				IF NOT bManualZIsSafe THEN
					TManualCmd.aTAxis[PA_X].Home.Enable := FALSE;
					TManualCmd.aTAxis[PA_Y].Home.Enable := FALSE;
					IF alrJogStep[PA_X] > lrManMaxXYMoveAllowed-0.1 THEN
						TManualCmd.aTAxis[PA_X].MoveBw.Enable := FALSE;
						TManualCmd.aTAxis[PA_X].MoveFw.Enable := FALSE;
					END_IF
					IF alrJogStep[PA_Y] > lrManMaxXYMoveAllowed-0.1 THEN
						TManualCmd.aTAxis[PA_Y].MoveBw.Enable := FALSE;
						TManualCmd.aTAxis[PA_Y].MoveFw.Enable := FALSE;
					END_IF
					IF alrJogStep[PA_Z1] > lrMaxXYMoveAllowed-0.1 THEN
						TManualCmd.aTAxis[PA_Z1].MoveFw.Enable := FALSE;
					END_IF
					IF alrJogStep[PA_Z2] > lrMaxXYMoveAllowed-0.1 THEN
						TManualCmd.aTAxis[PA_Z2].MoveFw.Enable := FALSE;
					END_IF
					TManualCmd.aTAxisPos[PA_X].MoveToTeach.Enable := TManualCmd.aTAxisPos[PA_X].MoveToTeach.Enable AND ABS(TManualCmd.aTAxisPos[PA_X].TeachedPos-aTRobotAxis[PA_X].lrCurrentPos) < lrManMaxXYMoveAllowed-0.1;
					TManualCmd.aTAxisPos[PA_Y].MoveToTeach.Enable := TManualCmd.aTAxisPos[PA_Y].MoveToTeach.Enable AND ABS(TManualCmd.aTAxisPos[PA_Y].TeachedPos-aTRobotAxis[PA_Y].lrCurrentPos) < lrManMaxXYMoveAllowed-0.1;
				END_IF
				bManInterlockOut := NOT bManualZIsSafe;
				TManualCmd.bWeightTableLeftValid := abWeightTableValid[PH_Left];
				TManualCmd.bWeightTableRightValid := abWeightTableValid[PH_Right];
				FOR i :=0 TO C_WEIGHT_TABLE_MAX DO
					TManualCmd.alrWeightTableLeft[i] := alrWeightTable[PH_Left,i];
					TManualCmd.alrWeightTableRight[i] := alrWeightTable[PH_Right,i];
				END_FOR
				FOR iSide:=0 TO 1 DO
					TManualCmd.TResetMotorUseTime[iSide].Enable := TRUE;
					TManualCmd.TResetSpindleUseTime[iSide].Enable := TRUE;
					TManualCmd.alrRatiog2mm[iSide] := alrRatiog2mm[iSide];
					TManualCmd.adwPearlsCounter[iSide] := adwPearlsCounter[iSide];
				END_FOR
				TManualCmd.lrWeightStepOnZ := lrLoadSensorStep;
				TManualCmd.aiDistanceSensor[0] := iContact1Distance;
				TManualCmd.aiDistanceSensor[1] := iContact2Distance;
				TManualCmd.iWeightSensor := iLoadSensorValue;
				CASE sCurrentState.eStep OF
					SP_ManualStp0 :
						FOR iSide:=0 TO 1 DO
							TManualCmd.aTEjectStick[iSide].Enable := TRUE;
							TManualCmd.aTActivateBlowing[iSide ].Enable := TRUE;
							TManualCmd.TActivateAspirationTable[iSide].Activate := abAspirationPearling[iSide];
							TManualCmd.aTStartMotor[iSide].Activate := abStartPearlingMotor[iSide];
							TManualCmd.aTOpenChuck[iSide].Activate := abOpenChuck[iSide];
							TManualCmd.aTEjectStick[iSide].Activate := abActivateEject[iSide];
							TManualCmd.aTActivateBlowing[iSide].Activate := abActivateBlowing[iSide];
							abStartPearlingMotor[iSide] := FALSE;
							TManualCmd.TActivateAspirationTable[iSide].Enable := TRUE;
							TManualCmd.TActivateAspirationTable[iSide].Activate := abAspirationPearling[iSide];
							TManualCmd.aiSpindleSpeedSetpoint[iSide] := aiSpindleManualSpeed[iSide];
							TManualCmd.aTCalibrateWeight[iSide].Activate := FALSE;
							TManualCmd.aiMotorStartedTimeout[iSide] := aiMotorStartedTimeout[iSide];
							TManualCmd.aiMotorStoppedTimeout[iSide] := aiMotorStoppedTimeout[iSide];
							TManualCmd.TResetMotorUseTime[iSide].Activate := FALSE;
							TManualCmd.TResetSpindleUseTime[iSide].Activate := FALSE;
						END_FOR
						FOR iAxis := 0 TO 3 DO
							TManualCmd.aTAxis[iAxis].JogStep := alrJogStep[iAxis];
							TManualCmd.aTAxis[iAxis].Home.Activate := FALSE;
							TManualCmd.aTAxis[iAxis].MoveFw.Activate := FALSE;
							TManualCmd.aTAxis[iAxis].MoveBw.Activate := FALSE;
							TManualCmd.aTAxis[iAxis].Specific.Activate := FALSE;
							TManualCmd.aTAxisPos[iAxis].MoveToTeach.Activate := FALSE;
						END_FOR
						TManualCmd.iCurrentMotorMinTh := iMCRMinThCurrent;
						TManualCmd.iCurrentMotorWarnTh := iMCRWarnThCurrent;
						TManualCmd.iCurrentMotorMaxTh := iMCRMaxThCurrent;
						TManualCmd.TActivateAspirationSharpen.Enable := TRUE;
						TManualCmd.TActivateAspirationSharpen.Activate := bAspirationSharpenOn;
						TManualCmd.TSafe.Activate := FALSE;
						bCalibrationInProgress := FALSE;
						sCurrentState.eStep := SP_ManualStp1;
					SP_ManualStp1:
						IF bStopReq THEN
							sCurrentState.eStatus := MS_Stopped;
						ELSE
							FOR iSide := 0 TO 1 DO
								abStartPearlingMotor[iSide] := TManualCmd.aTStartMotor[iSide].Activate;
								IF TManualCmd.TResetMotorUseTime[iSide].Activate THEN
									aTMotorCounter[iSide](bReset := TRUE);
									TManualCmd.TResetMotorUseTime[iSide].Activate := FALSE;
								END_IF
								IF TManualCmd.TResetSpindleUseTime[iSide].Activate THEN
									aTSpindleCounter[iSide](bReset := TRUE);
									TManualCmd.TResetSpindleUseTime[iSide].Activate := FALSE;
								END_IF
								IF TManualCmd.aiSpindleSpeedSetpoint[iSide] <> aiSpindleManualSpeed[iSide] THEN
									aiSpindleManualSpeed[iSide] := TManualCmd.aiSpindleSpeedSetpoint[iSide];
								END_IF
								IF TManualCmd.aiMotorStartedTimeout[iSide] <> aiMotorStartedTimeout[iSide] THEN
									aiMotorStartedTimeout[iSide] := TManualCmd.aiMotorStartedTimeout[iSide];
								END_IF
								IF TManualCmd.aiMotorStoppedTimeout[iSide] <> aiMotorStoppedTimeout[iSide] THEN
									aiMotorStoppedTimeout[iSide] := TManualCmd.aiMotorStoppedTimeout[iSide];
								END_IF
								// Calibration
								IF TManualCmd.aTCalibrateWeight[iSide].Activate THEN
									TManualCmd.aTCalibrateWeight[iSide].Activate := FALSE;
									bCalibrationInProgress := TRUE;
									iCurrentManAxis := iSide;
									sCurrentState.eStep := SP_ManualStp20;
								END_IF
							END_FOR
							IF TManualCmd.iCurrentMotorMinTh <> iMCRMinThCurrent THEN
								iMCRMinThCurrent := TManualCmd.iCurrentMotorMinTh;
							END_IF
							IF TManualCmd.iCurrentMotorMaxTh <> iMCRMaxThCurrent THEN
								iMCRMaxThCurrent := TManualCmd.iCurrentMotorMaxTh;
							END_IF
							IF TManualCmd.iCurrentMotorWarnTh <> iMCRWarnThCurrent THEN
								iMCRWarnThCurrent := TManualCmd.iCurrentMotorWarnTh;
							END_IF
							FOR iAxis := 0 TO 3 DO
								TManualCmd.aTAxisPos[iAxis].TeachedPos := alrRobotPos[iAxis,TManualCmd.e_TeachPos];
								IF TManualCmd.aTAxisPos[iAxis].Teach THEN
									alrRobotPos[iAxis,TManualCmd.e_TeachPos] := aTRobotAxis[iAxis].lrCurrentPos;
								END_IF
								TManualCmd.aTAxisPos[iAxis].Teach := FALSE;
							END_FOR
							FOR iAxis := 0 TO 3 DO
								IF (alrJogStep[iAxis] <> TManualCmd.aTAxis[iAxis].JogStep) THEN
									alrJogStep[iAxis] := TManualCmd.aTAxis[iAxis].JogStep;
								END_IF
								IF TManualCmd.aTAxisPos[iAxis].MoveToTeach.Activate THEN
									alrTargetPos[iAxis] := TManualCmd.aTAxisPos[iAxis].TeachedPos;
									iCurrentManAxis := iAxis;
									sCurrentState.eStep := SP_ManualStp2;
									EXIT;
								END_IF
								IF TManualCmd.aTAxis[iAxis].MoveFw.Activate THEN
									alrTargetPos[iAxis] := aTRobotAxis[iAxis].lrCurrentPos + alrJogStep[iAxis];
									iCurrentManAxis := iAxis;
									sCurrentState.eStep := SP_ManualStp2;
									EXIT;
								END_IF
								IF TManualCmd.aTAxis[iAxis].MoveBw.Activate THEN
									alrTargetPos[iAxis] := aTRobotAxis[iAxis].lrCurrentPos - alrJogStep[iAxis];
									iCurrentManAxis := iAxis;
									sCurrentState.eStep := SP_ManualStp2;
									EXIT;
								END_IF
								IF TManualCmd.aTAxis[iAxis].Home.Activate THEN
									iCurrentManAxis := iAxis;
									sCurrentState.eStep := SP_ManualStp40;
									EXIT;
								END_IF
							END_FOR
							IF TManualCmd.aTAxis[2].Specific.Activate THEN
								alrTargetPos[PA_Z1] := alrSafePos[PA_Z1];
								iCurrentManAxis := 2;
								sCurrentState.eStep := SP_ManualStp2;
							END_IF
							IF TManualCmd.aTAxis[3].Specific.Activate THEN
								alrTargetPos[PA_Z2] := alrSafePos[PA_Z2];
								iCurrentManAxis := 3;
								sCurrentState.eStep := SP_ManualStp2;
							END_IF
							IF TManualCmd.TSafe.Activate AND  (sCurrentState.eStep = SP_ManualStp1) THEN
								TManualCmd.TSafe.Activate := FALSE;
								sCurrentState.eStep := SP_ManualStp10;
							END_IF
							IF (sCurrentState.eStep = SP_ManualStp1) AND NOT bBypassMCR THEN
								sCurrentState.eStep := SP_ManualStp45;
							END_IF
						END_IF
					SP_ManualStp2:
						aeMoveRobotCommand[iCurrentManAxis] := AC_MoveAtAbsPos;
						sCurrentState.eStep := SP_ManualStp3;
					SP_ManualStp3:
						(* Wait until position is reached *)
						IF (aTRobotAxis[iCurrentManAxis].eCurrentState = AS_InPosition) THEN
							TManualCmd.aTAxisPos[iCurrentManAxis].MoveToTeach.Activate := FALSE;
							TManualCmd.aTAxis[iCurrentManAxis].Home.Activate := FALSE;
							TManualCmd.aTAxis[iCurrentManAxis].MoveFw.Activate := FALSE;
							TManualCmd.aTAxis[iCurrentManAxis].MoveBw.Activate := FALSE;
							TManualCmd.aTAxis[iCurrentManAxis].Specific.Activate := FALSE;
							sCurrentState.eStep := SP_ManualStp1;
						END_IF
					SP_ManualStp10: (*Move  Z1 and Z2 to Limit*)
						aeMoveRobotCommand[PA_Z1] := AC_MoveLimitNeg;
						aeMoveRobotCommand[PA_Z2] := AC_MoveLimitNeg;
						sCurrentState.eStep := SP_ManualStp11;
					SP_ManualStp11:
						IF aTRobotAxis[PA_Z1].eCurrentState= AS_OnLimitNeg AND aTRobotAxis[PA_Z2].eCurrentState= AS_OnLimitNeg THEN
							sCurrentState.eStep := SP_ManualStp12;
						ELSIF (aTRobotAxis[PA_Z1].eCurrentState= AS_OnLimitNeg AND aTRobotAxis[PA_Z2].eCurrentState = AS_InError) OR
							    (aTRobotAxis[PA_Z1].eCurrentState= AS_InError AND aTRobotAxis[PA_Z2].eCurrentState = AS_OnLimitNeg) OR
							    (aTRobotAxis[PA_Z1].eCurrentState= AS_InError AND aTRobotAxis[PA_Z2].eCurrentState = AS_InError) THEN
							sCurrentState.eStep := SP_ManualStp1;
						END_IF
					SP_ManualStp12: (* Init X/Y  *)
						aeMoveRobotCommand[PA_X] := AC_Init;
						aeMoveRobotCommand[PA_Y] := AC_Init;
						sCurrentState.eStep := SP_ManualStp13;
					SP_ManualStp13:
						IF aTRobotAxis[PA_X].eCurrentState= AS_InPosition AND aTRobotAxis[PA_Y].eCurrentState = AS_InPosition THEN
							sCurrentState.eStep := SP_ManualStp14;
						ELSIF (aTRobotAxis[PA_X].eCurrentState= AS_InPosition AND aTRobotAxis[PA_Y].eCurrentState = AS_InError) OR
								(aTRobotAxis[PA_X].eCurrentState= AS_InError AND aTRobotAxis[PA_Y].eCurrentState = AS_InPosition) OR
								(aTRobotAxis[PA_X].eCurrentState= AS_InError AND aTRobotAxis[PA_Y].eCurrentState = AS_InError) THEN
							sCurrentState.eStep := SP_ManualStp1;
						END_IF
					SP_ManualStp14: (* Move X/Y *)
						aeMoveRobotCommand[PA_X] := AC_MoveAtAbsPos;
						aeMoveRobotCommand[PA_Y] := AC_MoveAtAbsPos;
						alrTargetPos[PA_X] := alrSafePos[PA_X];
						alrTargetPos[PA_Y] := alrSafePos[PA_Y];
						sCurrentState.eStep := SP_ManualStp15;
					SP_ManualStp15:
						IF aTRobotAxis[PA_X].eCurrentState= AS_InPosition AND aTRobotAxis[PA_Y].eCurrentState = AS_InPosition THEN
							sCurrentState.eStep := SP_ManualStp16;
						ELSIF (aTRobotAxis[PA_X].eCurrentState= AS_InPosition AND aTRobotAxis[PA_Y].eCurrentState = AS_InError) OR
								(aTRobotAxis[PA_X].eCurrentState= AS_InError AND aTRobotAxis[PA_Y].eCurrentState = AS_InPosition) OR
								(aTRobotAxis[PA_X].eCurrentState= AS_InError AND aTRobotAxis[PA_Y].eCurrentState = AS_InError) THEN
							sCurrentState.eStep := SP_ManualStp1;
						END_IF
					SP_ManualStp16: (* Init Z1 and Z2*)
						aeMoveRobotCommand[PA_Z1] := AC_Init;
						aeMoveRobotCommand[PA_Z2] := AC_Init;
						sCurrentState.eStep := SP_ManualStp17;
					SP_ManualStp17:
						IF aTRobotAxis[PA_Z1].eCurrentState= AS_InPosition AND aTRobotAxis[PA_Z2].eCurrentState = AS_InPosition THEN
							sCurrentState.eStep := SP_ManualStp18;
						ELSIF (aTRobotAxis[PA_Z1].eCurrentState= AS_InPosition AND aTRobotAxis[PA_Z2].eCurrentState = AS_InError) OR
								(aTRobotAxis[PA_Z1].eCurrentState= AS_InError AND aTRobotAxis[PA_Z2].eCurrentState = AS_InPosition) OR
								(aTRobotAxis[PA_Z1].eCurrentState= AS_InError AND aTRobotAxis[PA_Z2].eCurrentState = AS_InError) THEN
							sCurrentState.eStep := SP_ManualStp1;
						END_IF
					SP_ManualStp18: (* Move up Z1 and Z2 *)
						aeMoveRobotCommand[PA_Z1] := AC_MoveAtAbsPos;
						aeMoveRobotCommand[PA_Z2] := AC_MoveAtAbsPos;
						alrTargetPos[PA_Z1] := alrSafePos[PA_Z1];
						alrTargetPos[PA_Z2] := alrSafePos[PA_Z2];
						sCurrentState.eStep := SP_ManualStp19;
					SP_ManualStp19:
						IF (aTRobotAxis[PA_Z1].eCurrentState= AS_InPosition OR aTRobotAxis[PA_Z1].eCurrentState = AS_InError) AND
								(aTRobotAxis[PA_Z2].eCurrentState= AS_InPosition OR aTRobotAxis[PA_Z2].eCurrentState = AS_InError) THEN
							sCurrentState.eStep := SP_ManualStp1;
						END_IF
					SP_ManualStp20:	 (* Do calibration *)
						abStartPearlingMotor[iCurrentManAxis] := FALSE;
						TManualCmd.aTStartMotor[iSide].Activate := FALSE;
						abWeightTableValid[iCurrentManAxis] := FALSE;
						FOR iSide := 0 TO 1 DO		// put the 2 brushes at Z safe position
							alrTargetPos[PA_Z1+iSide] := alrSafePos[PA_Z1+iSide];
							aeMoveRobotCommand[PA_Z1+iSide] := AC_MoveAtAbsPos;
						END_FOR
						sCurrentState.eStep := SP_ManualStp21;
					SP_ManualStp21:
						(* Wait until position is reached *)
						//IF (aTRobotAxis[PA_Z1+iCurrentManAxis].eCurrentState = AS_InPosition) AND aTWaitMotorStopped[iCurrentManAxis].Q THEN
						IF (aTRobotAxis[PA_Z1].eCurrentState = AS_InPosition) AND (aTRobotAxis[PA_Z2].eCurrentState = AS_InPosition) AND aTWaitMotorStopped[iCurrentManAxis].Q THEN
							aTStickContactValidated[iCurrentManAxis](IN := FALSE);
							alrLoadSensorOffset[iCurrentManAxis] := iLoadSensorValue;
							aeProbingArea[iCurrentManAxis] := PA_WeightCalibration;
							(* Move to load sensor position *)
							alrTargetPos[PA_X] := alrRobotPos[PA_X, PTP_WeightCalibrationPosZ1+iCurrentManAxis];
							alrTargetPos[PA_Y] := alrRobotPos[PA_Y, PTP_WeightCalibrationPosZ1+iCurrentManAxis];
							aeMoveRobotCommand[PA_X] := AC_MoveAtAbsPos;
							aeMoveRobotCommand[PA_Y] := AC_MoveAtAbsPos;
							sCurrentState.eStep := SP_ManualStp22;
						END_IF
					SP_ManualStp22:
						IF (eRobotXYStatus = AS_InPosition) THEN
							aTStickContactValidated[iCurrentManAxis](IN := TRUE,PT := TStickContactValidTime);
							IF aTStickContactValidated[iCurrentManAxis].Q THEN
								(* Get sensor threshold before getting down, so we can detetced if there is a stick *)
								aiContactThresholdArea[iCurrentManAxis , aeProbingArea[iCurrentManAxis]] := aiContactDistance[iCurrentManAxis];
								alrProbingLimit[iCurrentManAxis] :=  alrRobotPos[PA_Z1+iCurrentManAxis, PTP_WeightCalibrationPosZ1+iCurrentManAxis] + 0.5;
								alrTargetPos[PA_Z1+iCurrentManAxis] := alrRobotPos[PA_Z1+iCurrentManAxis, PTP_WeightCalibrationPosZ1+iCurrentManAxis];
								aeMoveRobotCommand[PA_Z1+iCurrentManAxis] := AC_MoveAtAbsPos;
								sCurrentState.eStep := SP_ManualStp23;
							END_IF
						END_IF
					SP_ManualStp23:
						(* Continuous move probing with analog sensor *)
						IF (aTRobotAxis[PA_Z1+ iCurrentManAxis].eCurrentState = AS_InPosition) THEN
							(* Move 0.5 mm above probing pos to check default sensor value *)
							alrTargetPos[PA_Z1 + iCurrentManAxis] := alrTargetPos[PA_Z1 + iCurrentManAxis] - 0.5;
							alrCurrentSpeed[PA_Z1 + iCurrentManAxis] := alrMaxRobotSpeed[PA_Z1 + iCurrentManAxis];
							aeMoveRobotCommand[PA_Z1 + iCurrentManAxis] := AC_MoveAtAbsPos;
							aTStickContactValidated[iCurrentManAxis](IN := FALSE);
							sCurrentState.eStep := SP_ManualStp24;
						ELSIF (aiContactDistance[iCurrentManAxis] > aiContactThresholdArea[iCurrentManAxis , aeProbingArea[iCurrentManAxis]] + alrSensorRate[iCurrentManAxis] * 0.5) THEN
							(* Stick is present, abort the process *)
							aeMoveRobotCommand[PA_Z1+iCurrentManAxis] := AC_Stop;
							bSecurityError := TRUE;
							iDebugPos := 6;
							iDebugSide := iCurrentManAxis;
							bCalibrationInProgress := FALSE;
							sCurrentState.eStep := SP_ManualStp1;
						END_IF
					SP_ManualStp24:
						IF (aTRobotAxis[PA_Z1 + iCurrentManAxis].eCurrentState = AS_InPosition) THEN
							aTStickContactValidated[iCurrentManAxis](IN := TRUE,PT := TStickContactValidTime);
							IF aTStickContactValidated[iCurrentManAxis].Q THEN
								aiContactThresholdArea[iCurrentManAxis , aeProbingArea[iCurrentManAxis]] := aiContactDistance[iCurrentManAxis];
								(* Move down slowly until we get contact *)
								alrTargetPos[PA_Z1 + iCurrentManAxis] := alrProbingLimit[iCurrentManAxis];
								alrCurrentSpeed[PA_Z1 + iCurrentManAxis] := lrSensorZSpeed;
								aeMoveRobotCommand[PA_Z1 + iCurrentManAxis] := AC_MoveAtAbsPos;
								sCurrentState.eStep := SP_ManualStp25;
							END_IF
						END_IF
					SP_ManualStp25:
						IF (aiContactDistance[iCurrentManAxis] >aiContactThresholdArea[iCurrentManAxis , aeProbingArea[iCurrentManAxis]] + alrSensorRate[iCurrentManAxis] * lrProbingThreshold) THEN
							aTStickContactValidated[iCurrentManAxis](IN := FALSE);
							aeMoveRobotCommand[PA_Z1 + iCurrentManAxis] := AC_Stop;
							sCurrentState.eStep := SP_ManualStp26;
						ELSIF (aTRobotAxis[PA_Z1 + iCurrentManAxis].eCurrentState = AS_InPosition) THEN
							aeMoveRobotCommand[PA_Z1+iCurrentManAxis] := AC_Stop;
							bSecurityError := TRUE;
							iDebugPos := 7;
							iDebugSide := iCurrentManAxis;
							bCalibrationInProgress := FALSE;
							sCurrentState.eStep := SP_ManualStp1;
						END_IF
					SP_ManualStp26:
						IF (aTRobotAxis[PA_Z1 + iCurrentManAxis].eCurrentState = AS_InPosition) THEN
							aTStickContactValidated[iCurrentManAxis](IN := TRUE,PT := TStickContactValidTime);
							IF aTStickContactValidated[iCurrentManAxis].Q THEN
								alrProbingPos[iCurrentManAxis] := aTRobotAxis[PA_Z1 + iCurrentManAxis].lrCurrentPos - (aiContactDistance[iCurrentManAxis] - aiContactThresholdArea[iCurrentManAxis , aeProbingArea[iCurrentManAxis]])/alrSensorRate[iCurrentManAxis];
								(* Move 2 mm above probing pos to check 1st measure *)
								alrTargetPos[PA_Z1 + iCurrentManAxis] := aTRobotAxis[PA_Z1 + iCurrentManAxis].lrCurrentPos - 2;
								alrCurrentSpeed[PA_Z1 + iCurrentManAxis] := alrMaxRobotSpeed[PA_Z1 + iCurrentManAxis];
								aeMoveRobotCommand[PA_Z1 + iCurrentManAxis] := AC_MoveAtAbsPos;
								sCurrentState.eStep := SP_ManualStp27;
							END_IF
						END_IF
					SP_ManualStp27:
						IF (aTRobotAxis[PA_Z1 + iCurrentManAxis].eCurrentState = AS_InPosition) THEN
							(* Move to contact position *)
							alrTargetPos[PA_Z1 + iCurrentManAxis] := alrTargetPos[PA_Z1 + iCurrentManAxis]+2;
							aeMoveRobotCommand[PA_Z1 + iCurrentManAxis] := AC_MoveAtAbsPos;
							aTStickContactValidated[iCurrentManAxis](IN := FALSE);
							sCurrentState.eStep := SP_ManualStp28;
						END_IF
					SP_ManualStp28:
						IF (aTRobotAxis[PA_Z1 + iCurrentManAxis].eCurrentState = AS_InPosition) THEN
							aTStickContactValidated[iCurrentManAxis](IN := TRUE,PT := TStickContactValidTime);
							IF aTStickContactValidated[iCurrentManAxis].Q THEN
								alrCheckProbingPos[iCurrentManAxis] := aTRobotAxis[PA_Z1 + iCurrentManAxis].lrCurrentPos - (aiContactDistance[iCurrentManAxis] - aiContactThresholdArea[iCurrentManAxis , aeProbingArea[iCurrentManAxis]])/alrSensorRate[iCurrentManAxis];
								IF (ABS(alrProbingPos[iCurrentManAxis] - alrCheckProbingPos[iCurrentManAxis]) < 0.05) AND (ABS(alrProbingPos[iCurrentManAxis] -  alrRobotPos[PA_Z1+iCurrentManAxis, PTP_WeightCalibrationPosZ1+iCurrentManAxis]) < 0.5) THEN
									sCurrentState.eStep := SP_ManualStp29;
								ELSE
									bSecurityError := TRUE;
									iDebugPos := 8;
									iDebugSide := iCurrentManAxis;
									bCalibrationInProgress := FALSE;
									sCurrentState.eStep := SP_ManualStp1;
								END_IF
							END_IF
						END_IF
					SP_ManualStp29:
						aTStickContactValidated[iCurrentManAxis](IN := FALSE);
						iTableIndex := 0;
						lrBasePos := alrProbingPos[iCurrentManAxis] - lrWeightCalibrationStartOffsetZ;
						alrTargetPos[PA_Z1+iCurrentManAxis] := lrBasePos;
						alrCurrentSpeed[PA_Z1+iCurrentManAxis] := lrSensorZSpeed;
						aeMoveRobotCommand[PA_Z1+iCurrentManAxis] := AC_MoveAtAbsPos;
						sCurrentState.eStep := SP_ManualStp30;
					SP_ManualStp30:
						IF (aTRobotAxis[PA_Z1+iCurrentManAxis].eCurrentState = AS_InPosition) THEN
							(* Measure delta contact position*)
							aTStickContactValidated[iCurrentManAxis](IN := TRUE,PT := TStickContactValidTime);
							IF aTStickContactValidated[iCurrentManAxis].Q THEN
								alrWeightTable[iCurrentManAxis,iTableIndex] := (INT_TO_LREAL(iLoadSensorValue) - alrLoadSensorOffset[iCurrentManAxis]) / lrLoadSensorRate;
								IF (iTableIndex < C_WEIGHT_TABLE_MAX) THEN
									iTableIndex := iTableIndex+1;
									alrTargetPos[PA_Z1+iCurrentManAxis] := lrBasePos + INT_TO_LREAL(iTableIndex)*lrLoadSensorStep;
									aeMoveRobotCommand[PA_Z1+iCurrentManAxis] := AC_MoveAtAbsPos;
									aTStickContactValidated[iCurrentManAxis](IN := FALSE);
								ELSE
									(* Calculate g to mm ratio *)
									alrRatiog2mm[iCurrentManAxis] := 1/((alrWeightTable[iCurrentManAxis,C_WEIGHT_TABLE_MAX] - alrWeightTable[iCurrentManAxis,10])/((C_WEIGHT_TABLE_MAX - 10)*lrLoadSensorStep));
									(* Move up to safe *)
									alrTargetPos[PA_Z1+iCurrentManAxis] := alrSafePos[PA_Z1+iCurrentManAxis];
									alrCurrentSpeed[PA_Z1+iCurrentManAxis] := alrMaxRobotSpeed[PA_Z1+iCurrentManAxis];
									aeMoveRobotCommand[PA_Z1+iCurrentManAxis] := AC_MoveAtAbsPos;
									sCurrentState.eStep := SP_ManualStp31;
								END_IF
							END_IF
						END_IF
					SP_ManualStp31:
						IF (aTRobotAxis[PA_Z1+iCurrentManAxis].eCurrentState = AS_InPosition) THEN
							abWeightTableValid[iCurrentManAxis] := TRUE;
							bCalibrationInProgress := FALSE;
							sCurrentState.eStep := SP_ManualStp1;
						END_IF
					SP_ManualStp40 : (* Init axis *)
						aeMoveRobotCommand[iCurrentManAxis] := AC_Home;
						sCurrentState.eStep := SP_ManualStp41;
					SP_ManualStp41 : (* Rotate the turn over to go to index position *)
						CASE aTRobotAxis[iCurrentManAxis].eCurrentState OF
							AS_InPosition, AS_InError:
								FOR iAxis := 0 TO 4 DO
									TManualCmd.aTAxis[iCurrentManAxis].Home.Activate := FALSE;
									TManualCmd.aTAxis[iCurrentManAxis].MoveFw.Activate := FALSE;
									TManualCmd.aTAxis[iCurrentManAxis].MoveBw.Activate := FALSE;
								END_FOR
								sCurrentState.eStep := SP_ManualStp1;
						END_CASE
					SP_ManualStp45:
						IF bMCRReady THEN
							yMCRChannel := 1;
							sCurrentState.eStep := SP_ManualStp46;
						END_IF
					SP_ManualStp46:
						(* Read speed *)
						eMCRCommand := MCRC_ReadSpeed;
						sCurrentState.eStep := SP_ManualStp47;
					SP_ManualStp47:
						IF bMCRReady THEN
							TManualCmd.aiMotorSpeed[yMCRChannel-1] := TMCRDrv.iSpeed;
							IF yMCRChannel = 1 THEN
								yMCRChannel := 2;
								sCurrentState.eStep := SP_ManualStp46;
							ELSE
								yMCRChannel := 1;
								sCurrentState.eStep := SP_ManualStp48;
							END_IF
						END_IF
					SP_ManualStp48:
						(* Read current *)
						eMCRCommand := MCRC_ReadCurrent;
						sCurrentState.eStep := SP_ManualStp49;
					SP_ManualStp49:
						IF bMCRReady THEN
							TManualCmd.arMotorCurrent[yMCRChannel-1] := LREAL_TO_REAL(TMCRDrv.lrCurrent);
							IF yMCRChannel = 1 THEN
								yMCRChannel := 2;
								sCurrentState.eStep := SP_ManualStp48;
							ELSE
								yMCRChannel := 1;
								sCurrentState.eStep := SP_ManualStp50;
							END_IF
						END_IF
					SP_ManualStp50:
						(* Set Ratio*)
						eMCRCommand := MCRC_SetRatio;
						TMCRDrv.lrRatio := asStickDataMMI[yMCRChannel - 1].lrMCRRatio;
						sCurrentState.eStep := SP_ManualStp51;
					SP_ManualStp51:
						IF bMCRReady THEN
							IF yMCRChannel = 1 THEN
								yMCRChannel := 2;
								sCurrentState.eStep := SP_ManualStp50;
							ELSE
								yMCRChannel := 1;
								sCurrentState.eStep := SP_ManualStp52;
							END_IF
						END_IF
					SP_ManualStp52:
						(* Set Speed*)
						eMCRCommand := MCRC_SetSpeed;
						TMCRDrv.iSpeedSetpoint := TManualCmd.aiSpindleSpeedSetpoint[yMCRChannel - 1];
						sCurrentState.eStep := SP_ManualStp53;
					SP_ManualStp53:
						IF bMCRReady THEN
							IF yMCRChannel = 1 THEN
								yMCRChannel := 2;
								sCurrentState.eStep := SP_ManualStp52;
							ELSE
								yMCRChannel := 1;
								sCurrentState.eStep := SP_ManualStp54;
							END_IF
						END_IF
					SP_ManualStp54:
						(* Set Parameter*)
						eMCRCommand := MCRC_SetParam;
						TMCRDrv.iOffsetCurrent := iMCROffsetCurrent[yMCRChannel - 1];
						TMCRDrv.iCurrentRatio := iMCRCurrentRatio[yMCRChannel - 1];
						sCurrentState.eStep := SP_ManualStp55;
					SP_ManualStp55:
						IF bMCRReady THEN
							IF yMCRChannel = 1 THEN
								yMCRChannel := 2;
								sCurrentState.eStep := SP_ManualStp54;
							ELSE
								yMCRChannel := 1;
								sCurrentState.eStep := SP_ManualStp1;
							END_IF
						END_IF
				END_CASE
				FOR iSide := 0 TO 1 DO
					abOpenChuck[iSide] := TManualCmd.aTOpenChuck[iSide].Activate;
					abActivateEject[iSide] := TManualCmd.aTEjectStick[iSide].Activate;
					abActivateBlowing[iSide] := TManualCmd.aTActivateBlowing[iSide].Activate;
					abAspirationPearling[iSide] := TManualCmd.TActivateAspirationTable[iSide].Activate;
				END_FOR
				bAspirationSharpenOn := TManualCmd.TActivateAspirationSharpen.Activate;
			MS_Paused:
				IF bStopReq THEN
					sCurrentState.eStatus := MS_Ready;
					sCurrentState.eStep := SP_RunStp1;
				END_IF
		END_CASE
	MC_Init :
		IF sCurrentState.bInitDone THEN
			sCurrentState.eStep := SP_InitStp50;
		ELSE
			sCurrentState.eStep := SP_InitStp1;
		END_IF
		sCurrentState.eStatus := MS_Init;
	MC_Run :
		IF (sCurrentState.eStep = SP_RunStp91) THEN
			sCurrentState.eStep := SP_RunStp92;
		END_IF
		sCurrentState.eStatus := MS_Running;
	MC_Manual :
		sCurrentState.bInitDone := FALSE;
		sCurrentState.eStatus := MS_Manual;
		sCurrentState.eStep := SP_ManualStp0;
	MC_Stop :
		//eMCRCommand := MCRC_UpdateMemory;				// TODO : HFO, Problème de comunication, impossible de mettre à jour les chips, controle si ok?
		sCurrentState.eStatus := MS_Stopped;
END_CASE;

(* The pearling motor doesn't run if not in production *)
IF (sCurrentState.eStatus <> MS_Running) AND (sCurrentState.eStatus <> MS_Manual) THEN
	FOR iSide := 0 TO 1 DO
		abStartPearlingMotor[iSide] := FALSE;
		abActivateBlowing[iSide] := FALSE;
	END_FOR
END_IF
IF (sCurrentState.eStatus = MS_Running) THEN
	FOR iSide:=0 TO 1 DO
		(* Force motor running if possible *)
		IF NOT abDoProbing[iSide] AND NOT abChangeStick[iSide]  AND NOT  abSharpenStick[iSide] AND abChuckClosed[iSide] AND
				((sCurrentState.eStep < SP_RunStp30) OR
				(sCurrentState.eStep > SP_RunStp33)) THEN
			IF bKeepBothHeadWarm THEN
				abStartPearlingMotor[iSide] := TRUE;
			ELSE
				abStartPearlingMotor[iSide] := abUseSpindle[iSide];
			END_IF
		END_IF
	END_FOR
	FOR iSide:=0 TO 1 DO
		abActivateBlowing[iSide] := abStartPearlingMotor[PH_Left] OR abStartPearlingMotor[PH_Right]; (* Activate blowing if at least one head is pearling *)
	END_FOR
END_IF

IF bResetErrors THEN
	sCurrentState.bInError := FALSE;
END_IF

(* Define dynamics *)

FOR iAxis:=0 TO 3 DO
	IF (aeMoveRobotCommand[iAxis] = AC_MoveAtAbsPos) THEN
		IF (ABS(aTRobotAxis[iAxis].lrCurrentPos - alrTargetPos[iAxis]) > 10) THEN
			alrDynParams[iAxis] := alrLowDynParams[iAxis];
		ELSE
			alrDynParams[iAxis] := alrHighDynParams[iAxis];
		END_IF
	END_IF
END_FOR


IF ((ABS(aTRobotAxis[PA_X].lrCurrentPos - alrTargetPos[PA_X]) > lrMaxXYMoveAllowed) AND (aeMoveRobotCommand[PA_X] <> AC_None)) OR
		((ABS(aTRobotAxis[PA_Y].lrCurrentPos - alrTargetPos[PA_Y]) > lrMaxXYMoveAllowed) AND (aeMoveRobotCommand[PA_Y] <> AC_None)) THEN
	IF (aTRobotAxis[PA_Z1].lrCurrentPos > (alrSafePos[PA_Z1] + lrSafeTolerance)) OR
			(aTRobotAxis[PA_Z2].lrCurrentPos > (alrSafePos[PA_Z2] + lrSafeTolerance)) THEN
		IF eStickStep<> SP_RunStp61 AND eStickStep<> SP_RunStp62 THEN
			aeMoveRobotCommand[PA_X] := AC_ForceStop;
			aeMoveRobotCommand[PA_Y] := AC_ForceStop;
			sCurrentState.bInitDone := FALSE;
			bSecurityError := TRUE;
			iDebugPos := 9;
			iDebugSide := -1;
		END_IF
	END_IF
END_IF

IF (sCurrentState.eStatus = MS_Manual) THEN
	FOR iAxis:=0 TO 3 DO
		IF bManualZIsSafe THEN
			alrCurrentSpeed[iAxis] := aTRobotAxis[iAxis].lrFastManualSpeed;
		ELSE
			alrCurrentSpeed[iAxis] :=  aTRobotAxis[iAxis].lrManualSpeed;
		END_IF
	END_FOR
END_IF

(* Robot command *)
aTRobotAxis[PA_X](
	eCommand 		:= aeMoveRobotCommand[PA_X],
	lrTargetPos 		:= alrTargetPos[PA_X],
	lrTargetSpeed 	:= alrCurrentSpeed[PA_X],
	lrAcceleration 	:= alrDynParams[PA_X].Acc,
	lrDeceleration 	:= alrDynParams[PA_X].Dec,
	lrJerk 			:= alrDynParams[PA_X].Jerk,
	sAxis		 	:= sXAxisRef,
	bHomeSensor 	:= bHomeX,
	eAxisType		:= AT_AX5000,
	bPowerIsOn		:= bPowerOn,
	bPosLimitSwitch	:= NOT bLimitPosX,
	bNegLimitSwitch	:= NOT bLimitNegX,
	lrMoveOutDist	:= 50,
	bResetErrors	 	:= bResetErrors,
	stServoButton		:= TManualCmd.aTAxis[PA_X].ServoON
);
aeMoveRobotCommand[PA_X] := AC_None;
bXAxisError := (aTRobotAxis[PA_X].eCurrentState = AS_InError);

aTRobotAxis[PA_Y](
	eCommand 		:= aeMoveRobotCommand[PA_Y],
	lrTargetPos 		:= alrTargetPos[PA_Y],
	lrTargetSpeed 	:= alrCurrentSpeed[PA_Y],
	lrAcceleration 	:= alrDynParams[PA_Y].Acc,
	lrDeceleration 	:= alrDynParams[PA_Y].Dec,
	lrJerk 			:= alrDynParams[PA_Y].Jerk,
	sAxis		 	:= sYAxisRef,
	bHomeSensor 	:= bHomeY,
	eAxisType		:= AT_AX5000,
	bPowerIsOn		:= bPowerOn,
	bPosLimitSwitch	:= NOT bLimitPosY,
	bNegLimitSwitch	:= NOT bLimitNegY,
	lrMoveOutDist	:= 50,
	bResetErrors	 	:= bResetErrors,
	stServoButton		:= TManualCmd.aTAxis[PA_Y].ServoON
);
aeMoveRobotCommand[PA_Y] := AC_None;
bYAxisError := (aTRobotAxis[PA_Y].eCurrentState = AS_InError);

aTRobotAxis[PA_Z1](
	eCommand 		:= aeMoveRobotCommand[PA_Z1],
	lrTargetPos 		:= alrTargetPos[PA_Z1],
	lrTargetSpeed 	:= alrCurrentSpeed[PA_Z1],
	lrAcceleration 	:= alrDynParams[PA_Z1].Acc,
	lrDeceleration 	:= alrDynParams[PA_Z1].Dec,
	lrJerk 			:= alrDynParams[PA_Z1].Jerk,
	sAxis		 	:= sZ1AxisRef,
	bHomeSensor 	:= bHomeZ1,
	bPosLimitSwitch	:= NOT bLimitPosZ1,
	bNegLimitSwitch	:= NOT bLimitNegZ1,
	eAxisType		:= AT_Standard,
	bPowerIsOn		:= bPowerOn,
	bResetErrors	 	:= bResetErrors,
	lrMoveOutDist	:= 10,
	stServoButton		:= TManualCmd.aTAxis[PA_Z1].ServoON
);
aeMoveRobotCommand[PA_Z1] := AC_None;
bZ1AxisError := (aTRobotAxis[PA_Z1].eCurrentState = AS_InError);

aTRobotAxis[PA_Z2](
	eCommand 		:= aeMoveRobotCommand[PA_Z2],
	lrTargetPos 		:= alrTargetPos[PA_Z2],
	lrTargetSpeed 	:= alrCurrentSpeed[PA_Z2],
	lrAcceleration 	:= alrDynParams[PA_Z2].Acc,
	lrDeceleration 	:= alrDynParams[PA_Z2].Dec,
	lrJerk 			:= alrDynParams[PA_Z2].Jerk,
	sAxis		 	:= sZ2AxisRef,
	bHomeSensor 	:= bHomeZ2,
	bPosLimitSwitch	:= NOT bLimitPosZ2,
	bNegLimitSwitch	:= NOT bLimitNegZ2,
	eAxisType		:= AT_Standard,
	bPowerIsOn		:= bPowerOn,
	bResetErrors	 	:= bResetErrors,
	lrMoveOutDist	:= 10,
	stServoButton		:= TManualCmd.aTAxis[PA_Z2].ServoON
);
aeMoveRobotCommand[PA_Z2] := AC_None;
bZ2AxisError := (aTRobotAxis[PA_Z2].eCurrentState = AS_InError);

(* Get move result *)
eRobotXYStatus := AS_Moving;
IF (aTRobotAxis[PA_X].eCurrentState = AS_InError) OR (aTRobotAxis[PA_Y].eCurrentState = AS_InError) THEN
	eRobotXYStatus := AS_InError;
ELSIF (aTRobotAxis[PA_X].eCurrentState = AS_InPosition) AND (aTRobotAxis[PA_Y].eCurrentState = AS_InPosition) THEN
		eRobotXYStatus := AS_InPosition;
END_IF

(* Check gripper error *)
aTCheckChuck[PH_Left](
	bJackGoOut	:= abOpenChuck[PH_Left],
	bJackIsIn	:= abChuckClosed[PH_Left],
	bJackIsOut	:= abChuckOpened[PH_Left],
	bResetErrors := bResetErrors,
	bJackError	=> bChuck1Error
);
aTCheckChuck[PH_Right](
	bJackGoOut	:= abOpenChuck[PH_Right],
	bJackIsIn	:= abChuckClosed[PH_Right],
	bJackIsOut	:= abChuckOpened[PH_Right],
	bResetErrors := bResetErrors,
	bJackError	=> bChuck2Error
);

TMCRDrv(
	iComPort			:= iComPort,
	yChannel			:= yMCRChannel,
	iMinCurrent			:= 5,
	iCheckTime			:= 10,
	bCommandExecuted	=> bMCRReady,
	bCommandError		=> bMCRError,
	eCommand			:= eMCRCommand,
	RxBuffer			:= sRecData,
	TxBuffer			:= sTransData,
	bReset				:= bResetErrors,
	ayChannelStatus		=> ayChannelStatus,

);

IF bBypassMCR THEN
	bMCRError := FALSE;
END_IF

(* Handle errors *)
IF bResetErrors THEN
	(* Reset all errors not related to controls *)
	FOR iSide := 0 TO 1 DO
		abSpindleError[iSide] := FALSE;
		abStickBroken[iSide] := FALSE;
		abMotorError[iSide] := FALSE;
		abCurrentReadError[iSide] := FALSE;
		abPearlingWeightOutOfToleranceError[iSide] := FALSE;
		abCurrentLimitWarning[iSide] := FALSE;
	END_FOR
	bSecurityError := FALSE;
	bStickNotTakenError := FALSE;
	bLeftSpindleUsedWarning := FALSE;
	bRightSpindleUsedWarning := FALSE;
	bLeftMotorUsedWarning := FALSE;
	bRightMotorUsedWarning := FALSE;
END_IF


IF bXAxisError OR bYAxisError OR bZ1AxisError OR bZ2AxisError OR bChuck1Error OR bChuck2Error OR abSpindleError[PH_Left] OR abSpindleError[PH_Right] OR bSecurityError OR bMCRError OR abMotorError[PH_Left] OR abMotorError[PH_Right] OR
		 ((abStickBroken[PH_Left] OR abStickBroken[PH_Right]) AND sStickDataShared.sStickDataMMIShared.bStopOnStickBreak) OR
		(( abPearlingWeightOutOfToleranceError[PH_Left] OR abPearlingWeightOutOfToleranceError[PH_Right]) AND sStickDataShared.sStickDataMMIShared.bStopOnWeightOutOfTolerance) THEN
	sCurrentState.bInError := TRUE;
	IF (sCurrentState.eStatus <> MS_Manual) AND (sCurrentState.eStatus <> MS_Stopped) AND (sCurrentState.eStatus <> MS_Init) THEN
		sCurrentState.eStatus := MS_Ready;
	END_IF
END_IF

IF NOT bPowerOn OR bXAxisError OR bYAxisError OR bZ1AxisError OR bZ2AxisError OR bSecurityError OR bMCRError THEN
	sCurrentState.bInitDone := FALSE;
	IF (sCurrentState.eStatus <> MS_Manual) THEN
		sCurrentState.eStatus := MS_Stopped;
	END_IF
END_IF


IF NOT bPowerOn OR bSecurityError THEN
	bClearZRef := TRUE;
END_IF

IF bClearZRef THEN
	FOR i:= 0 TO 3 DO
		FOR j:= 0 TO 1 DO
			FOR iSide := 0 TO 1 DO
				abZRefTaken[i, j, iSide] := FALSE;
			END_FOR
		END_FOR
	END_FOR
	bClearZRef := FALSE;
END_IF

(* Security *)
FOR iSide:=0 TO 1 DO
	IF abOpenChuck[iSide] OR NOT abChuckClosed[iSide] THEN
		abStartPearlingMotor[iSide] := FALSE;
	END_IF
	IF NOT abUseSpindle[iSide] AND  (sCurrentState.eStatus <> MS_Manual) THEN
		abStartPearlingMotor[iSide] := FALSE;
	END_IF
END_FOR

sCurrentState.bRunning := (sCurrentState.eStatus = MS_Running);
sCurrentState.bWarning := bLeftSpindleUsedWarning OR bRightSpindleUsedWarning OR bLeftMotorUsedWarning OR bRightMotorUsedWarning OR bRightSpindleLimitWarning;

bModuleError := sCurrentState.bInError;
IF (sCurrentState.eStatus <> MS_Running) THEN eRunStatus := RS_NotRunning; END_IF

TDebug.iStep := sCurrentState.eStep;
TDebug.iStickStep := eStickStep;
FOR iSide := 0 TO 1 DO
	TDebug.aiProbingStep[iSide] := aeProbingStep[iSide];
	TDebug.abOpenChuck[iSide] := abOpenChuck[iSide];
	TDebug.abSharpenStick[iSide] := abSharpenStick[iSide];
	TDebug.abChangeStick[iSide] := abChangeStick[iSide];
	TDebug.abUseSpindle[iSide] := abUseSpindle[iSide];
END_FOR

(* Handle motor and spindle running timers *)
FOR iSide := 0 TO 1 DO
	adwMotorRunningHours[iSide] := aTMotorCounter[iSide].dwHours;
	adwSpindleRunningHours[iSide] := aTSpindleCounter[iSide].dwHours;
	aTDetectSpindleCooled[iSide](IN := NOT abStartPearlingMotor[iSide], pt := T#60M);
	IF (aTDetectSpindleCooled[iSide].Q) THEN
		abNeedSpindleHeatOn[iSide] := TRUE;
	END_IF
	aTWaitSpindleHeatOn[iSide](IN := abStartPearlingMotor[iSide], pt := T#10M);
	IF (aTWaitSpindleHeatOn[iSide].Q) THEN
		abNeedSpindleHeatOn[iSide] := FALSE;
	END_IF
	IF (NOT abUseSpindle[iSide]) THEN
		abNeedSpindleHeatOn[iSide] := FALSE;
	END_IF
END_FOR
bLeftSpindleHeatWarning := abStartPearlingMotor[PH_Left] AND abNeedSpindleHeatOn[PH_Left];
bRightSpindleHeatWarning := abStartPearlingMotor[PH_Right] AND abNeedSpindleHeatOn[PH_Right];
(* Set motor/spindle warning only every hour *)
IF aTSpindleCounter[PH_Left].bHoursTrig THEN
	bLeftSpindleUsedWarning := (adwSpindleRunningHours[PH_Left] > dwMaxSpindleRunningHours);
END_IF
IF aTSpindleCounter[PH_Right].bHoursTrig THEN
	bRightSpindleUsedWarning := (adwSpindleRunningHours[PH_Right] > dwMaxSpindleRunningHours);
END_IF
IF aTMotorCounter[PH_Left].bHoursTrig THEN
	bLeftMotorUsedWarning := (adwMotorRunningHours[PH_Left] > dwMaxMotorRunningHours);
END_IF
IF aTMotorCounter[PH_Right].bHoursTrig THEN
	bRightMotorUsedWarning := (adwMotorRunningHours[PH_Right] > dwMaxMotorRunningHours);
END_IF

(* Optimize code *)
bStartPearlingMotor1 := abStartPearlingMotor[PH_Left];
bStartPearlingMotor2 := abStartPearlingMotor[PH_Right];
bOpenChuck1 := abOpenChuck[PH_Left];
bOpenChuck2 := abOpenChuck[PH_Right];
bActivateEject1 := abActivateEject[PH_Left];
bActivateEject2 := abActivateEject[PH_Right];
bSpindle1Error := abSpindleError[PH_Left];
bSpindle2Error := abSpindleError[PH_Right];
bStickContact1 := abStickContact[PH_Left];
bStickContact2 := abStickContact[PH_Right];
bActivateBlowing1 := abActivateBlowing[PH_Left];
bActivateBlowing2 := abActivateBlowing[PH_Right];
bCurrent1ReadError := abCurrentReadError[PH_Left];
bCurrent2ReadError := abCurrentReadError[PH_Right];
bMotor1Error := abMotorError[PH_Left];
bMotor2Error := abMotorError[PH_Right];
bAspirationPearling1On := abAspirationPearling[PH_Left];
bAspirationPearling2On := abAspirationPearling[PH_Right];
bStick1Broken := abStickBroken[PH_Left];
bStick2Broken := abStickBroken[PH_Right];
bPearlingWeight1OutOfToleranceError := abPearlingWeightOutOfToleranceError[PH_Left];
bPearlingWeight2OutOfToleranceError := abPearlingWeightOutOfToleranceError[PH_Right];
bLeftSpindleLimitWarning := abCurrentLimitWarning[PH_Left];
bRightSpindleLimitWarning := abCurrentLimitWarning[PH_Right];
atStickValidateTime[PH_Left] := TIME_TO_LREAL(aTStickContactValidated[PH_Left].ET);
atStickValidateTime[PH_Right] := TIME_TO_LREAL(aTStickContactValidated[PH_Right].ET);

ai_ProbingStep[0] := aeProbingStep[0];
ai_ProbingStep[1] := aeProbingStep[1];
i_StickStep := eStickStep;

END_FUNCTION_BLOCK

// ---- POUs/Drivers/MCRDrv.TcPOU
FUNCTION_BLOCK MCRDrv

(*
	Description 	: Function bloc to handle MCR board
	Author		: DRE
	Date		: 22.09.2016
	Version		: 1.00

	Modifications :

*)

VAR_INPUT
	iComPort				: INT;
	yChannel			: BYTE;
(*	iMinDiffCurrent		: INT; *)
	iMinThCurrent		: INT;
	iMaxThCurrent		: INT;
	iWarnThCurrent		: INT;
	iCheckTime			: INT;
	iMinCurrent			: INT;
	iSpeedSetpoint		: INT;
	lrRatio				: LREAL;
	bReset				: BOOL;
	iOffsetCurrent		: INT;
	iCurrentRatio		: INT;
	iMachineWO			: DINT;
	iMachineSN			: INT;
	yMachineSide		: BYTE;
END_VAR
VAR_OUTPUT
	bCommandExecuted	: BOOL					:= TRUE;
	bCommandError		: BOOL					:= FALSE;
	lrCurrent				: LREAL;
	lrPower				: LREAL;
	iSpeed				: INT;
	sVersion			: STRING;
	ayChannelStatus		: ARRAY[0..1] OF BYTE;
END_VAR
VAR_IN_OUT
	eCommand			: TMCRCommands;
	RxBuffer			: ComBuffer;
	TxBuffer			: ComBuffer;
END_VAR
VAR
	bFirstPass			: BOOL					:= TRUE;
(*	bConnect			: BOOL					:= FALSE;*)
	bSendBusy			: BOOL;
	bStringReceived		: BOOL;
	bReceivedBusy		: BOOL;
	bReceiveTimeout		: BOOL;
	SendErrorID			: ComError_t;
	ReceiveErrorID		: ComError_t;
	acSuffix				: STRING(255)			 := '$r';
	eStep				: INT					:= 1;
	strReceived			: STRING(255);
	strReceivedCh1			: STRING(255);
	strReceivedCh2			: STRING(255);
	lengthCh1			: INT := 2;
	lengthCh2			: INT := 2;
	posCh1			: INT	 := 2;
	posCh2			: INT	 := 4;
	SendString			: SendString;
	sString2Send			: STRING(255);
	ReceiveString		: ReceiveString;
	ClearComBuffer		: ClearComBuffer;
	bCanLog				: BOOL			:= FALSE;
	acLogText			: STRING(255);
	acLogFileName		: STRING(255);
	fbFormat 			: FB_FormatString;
	fbOpenFile			: FB_FileOpen;
	fbCloseFile			: FB_FileClose;
	fbWriteFile			: FB_FileWrite;
	hLogFile				: UINT;
	bOpenFile			: BOOL			:= FALSE;
	bCloseFile			: BOOL			:= FALSE;
	bWriteFile			: BOOL			:= FALSE;
	sTempString			: STRING(255);
	yCheckSum			: BYTE;
	sLastStringRec		: STRING(255);
	sCommandString		: STRING(255);
	TRecTimeout			: TON;
	iRatio				: INT;
	abWaitingForPower	: ARRAY[0..1] OF BOOL;
	alrPower			: ARRAY[0..1] OF LREAL;
	bFirstError 		: BOOL 			:= 	TRUE;
END_VAR

IF (bFirstPass) THEN
	ClearComBuffer(Buffer := RxBuffer);
	fbFormat(sFormat := 'C:\MPS_HMI\logs\test%.1d.log', arg1 := F_INT(iComPort), sOut => acLogFileName);
	bFirstPass := FALSE;
END_IF

fbOpenFile(
	sNetId			:= 	'',
	sPathName		:=	acLogFileName,
	nMode			:=	FOPEN_MODEAPPEND OR FOPEN_MODETEXT ,
	hFile			=>	hLogFile,
	bExecute		:=	bOpenFile
);
IF bOpenFile THEN
	bWriteFile := TRUE;
END_IF
bOpenFile := FALSE;

fbCloseFile (
	sNetId			:=	'',
	hFile			:=	hLogFile,
	bExecute		:=	bCloseFile
);
IF bCloseFile THEN
	bWriteFile := FALSE;
END_IF
bCloseFile := FALSE;

ReceiveString(
	Prefix			:= ,
	Suffix			:= acSuffix,
	Timeout			:= t#5s,
	Reset			:= ,
	ReceivedString	:= strReceived,
	RXbuffer			:= RxBuffer,
	StringReceived	=> bStringReceived,
	Busy			=> bReceivedBusy,
	Error			=> ReceiveErrorID,
	RxTimeout		=> bReceiveTimeout
);
IF (bStringReceived AND (ReceiveErrorID = COMERROR_NOERROR)) THEN
	sLastStringRec := strReceived;
	IF bWriteFile THEN
		bCanLog := TRUE;
		fbFormat(sFormat := '<--  %S$R$N', arg1 := F_STRING(strReceived), sOut => acLogText);
	END_IF
	IF (eStep = 1) THEN
		IF (LEFT(strReceived,2) = 'p1') AND abWaitingForPower[0] THEN
			IF (LEN(sLastStringRec) = 13) THEN
				alrPower[0] := STRING_TO_LREAL(MID(strReceived,7,4));
			ELSE
				bCommandError := TRUE;
			END_IF
			abWaitingForPower[0] := FALSE;
		ELSIF (LEFT(strReceived,2) = 'p1') AND abWaitingForPower[1] THEN
			IF (LEN(sLastStringRec) = 13) THEN
				alrPower[1] := STRING_TO_LREAL(MID(strReceived,7,4));
			ELSE
				bCommandError := TRUE;
			END_IF
			abWaitingForPower[1] := FALSE;
		END_IF
	END_IF
END_IF

CASE eStep OF
	1 : (* Check the command *)
		CASE eCommand OF
			MCRC_ConfigMeasure :
				fbFormat(sFormat := 'C%.1d,%.2d,%.3d', arg1 := F_BYTE(yChannel),arg2 := F_INT(iMinCurrent), arg3 := F_INT(iCheckTime), sOut => sTempString);
				eStep := 2;
			MCRC_ReadCurrent :
				fbFormat(sFormat := 'I%.1d', arg1 := F_BYTE(yChannel), sOut => sTempString);
				eStep := 2;
			MCRC_StartPower :
				fbFormat(sFormat := 'P%.1d', arg1 := F_BYTE(yChannel), sOut => sTempString);
				abWaitingForPower[yChannel-1] := TRUE;
				alrPower[yChannel-1] := 0;
				eStep := 2;
			MCRC_ReadSpeed :
				fbFormat(sFormat := 'S%.1d', arg1 := F_BYTE(yChannel), sOut => sTempString);
				eStep := 2;
			MCRC_GetPower :
				abWaitingForPower[yChannel-1] := FALSE;
				lrPower := alrPower[yChannel-1];
				bCommandExecuted := TRUE;
			MCRC_GetVersion :
				sTempString :=  'V';
				eStep := 2;
			MCRC_SetParam :
				IF(iOffsetCurrent < 0)THEN
					fbFormat(sFormat := 'W%.1d,%.4d,%.5d', arg1 := F_BYTE(yChannel),arg2 := F_INT(iOffsetCurrent), arg3 := F_INT(iCurrentRatio), sOut => sTempString);
				ELSE
					fbFormat(sFormat := 'W%.1d,%.5d,%.5d', arg1 := F_BYTE(yChannel),arg2 := F_INT(iOffsetCurrent), arg3 := F_INT(iCurrentRatio), sOut => sTempString);
				END_IF
				eStep := 2;
			MCRC_GetParam :
				fbFormat(sFormat := 'R%.1d', arg1 := F_BYTE(yChannel), sOut => sTempString);
				eStep := 2;
			MCRC_SetSpeed :
				fbFormat(sFormat := 'T%.1d,%.4d', arg1 := F_BYTE(yChannel), arg2 := F_INT(iSpeedSetpoint), sOut => sTempString);
				eStep := 2;
			MCRC_SetRatio:
				iRatio := LREAL_TO_INT(lrRatio*100.0);
				fbFormat(sFormat := 'D%.1d,%.4d', arg1 := F_BYTE(yChannel), arg2 := F_INT(iRatio), sOut => sTempString);
				eStep := 2;
			MCRC_UpdateMemory:
				sTempString :=  'K';
				eStep := 2;
			MCRC_DefineCurrentThr :
				fbFormat(sFormat := 'M%.1d,%.3d,%.3d,%.3d', arg1 := F_BYTE(yChannel), arg2 := F_INT(iMinThCurrent),  arg3 := F_INT(iMaxThCurrent),  arg4 := F_INT(iWarnThCurrent), sOut => sTempString);
				eStep := 2;
			MCRC_DefineMachineID :
				fbFormat(sFormat := 'X,%.6d%.3d%c', arg1 := F_DINT(iMachineWO), arg2 := F_INT(iMachineSN),  arg3 := F_BYTE(yMachineSide), sOut => sTempString);
				eStep := 2;
			MCRC_GetStatus :
				sTempString :=  'Z';
				eStep := 2;
		END_CASE
		IF (eStep = 2) THEN
			bCommandExecuted := FALSE;
			yCheckSum := yCalcCheckSum(sTempString);
			yCheckSum := 0;
			fbFormat(sFormat := '%s%.2x%s', arg1 := F_STRING(sTempString), arg2 := F_BYTE(yCheckSum), arg3 := F_STRING(acSuffix), sOut => sString2Send);
			SendString(
				SendString	:= sString2Send,
				TXbuffer		:= TxBuffer,
				Busy		=> bSendBusy,
				Error		=> SendErrorID);
			IF bWriteFile THEN
				bCanLog := TRUE;
				fbFormat(sFormat := '-->  %S$R$N', arg1 := F_STRING(sString2Send), sOut => acLogText);
			END_IF
		END_IF
	2 : (* Wait until the end of transmission *)
		IF (SendErrorID = 0) THEN
			IF NOT bSendBusy THEN
				IF (eCommand = MCRC_StartPower) THEN
					eStep := 1;
					bCommandExecuted := TRUE;
					eCommand := MCRC_None;
				ELSE
					TRecTimeout(IN := FALSE);
					eStep := 3;
				END_IF
			END_IF
		END_IF
	3: (* Wait for the answer *)
		TRecTimeout(IN := TRUE,PT := t#5s);
		IF (ReceiveErrorID = 0) AND NOT bReceiveTimeout THEN
			IF bStringReceived  THEN
				eStep := 4;
			END_IF
		END_IF
		IF TRecTimeout.Q THEN
			strReceived := '';
			bCanLog := TRUE;
			fbFormat(sFormat := '<--  Timeout', sOut => acLogText);
			eStep := 4;
		END_IF
	4 : (* Process the line *)
		(* First check if checksum is OK *)
		yCheckSum := yCalcCheckSum(LEFT(sLastStringRec,LEN(sLastStringRec)-3));
		sCommandString := LEFT(sLastStringRec,LEN(sLastStringRec)-3);
		fbFormat(sFormat := '%s%.2x%s', arg1 := F_STRING(sCommandString), arg2 := F_BYTE(yCheckSum), arg3 := F_STRING(acSuffix), sOut => sTempString);
		IF (sTempString = strReceived) THEN
			CASE eCommand OF
				MCRC_ConfigMeasure :
					fbFormat(sFormat := 'c%01d', arg1 := F_BYTE(yChannel), sOut => sTempString);
					IF (LEN(sLastStringRec) = 5) AND (LEFT(strReceived,2) = sTempString) THEN
						eStep := 1;
					ELSE
						eStep := 0; (* error *)
					END_IF
				MCRC_ReadCurrent :
					fbFormat(sFormat := 'i%01d,', arg1 := F_BYTE(yChannel), sOut => sTempString);
					lrCurrent := STRING_TO_LREAL(MID(sLastStringRec,6,4));
					IF (LEN(sLastStringRec) = 12) AND (LEFT(strReceived,3) = sTempString) THEN
						eStep := 1;
					ELSE
						eStep := 0; (* error *)
					END_IF
				MCRC_ReadSpeed :
					fbFormat(sFormat := 's%01d,', arg1 := F_BYTE(yChannel), sOut => sTempString);
					iSpeed := STRING_TO_INT(MID(sLastStringRec,4,4));
					IF (LEN(sLastStringRec) = 10) AND (LEFT(strReceived,3) = sTempString) THEN
						eStep := 1;
					ELSE
						eStep := 0; (* error *)
					END_IF
				MCRC_GetVersion :
					IF (LEN(sLastStringRec) = 10) AND (LEFT(strReceived,1) = 'v') THEN
						sVersion := MID(sLastStringRec,6,2);
						eStep := 1;
					ELSE
						eStep := 0; (* error *)
					END_IF
				MCRC_SetParam :
					fbFormat(sFormat := 'w%01d', arg1 := F_BYTE(yChannel), sOut => sTempString);
					IF (LEN(sLastStringRec) = 5) AND (LEFT(strReceived,2) = sTempString) THEN
						eStep := 1;
					ELSE
						eStep := 0; (* error *)
					END_IF
				MCRC_GetParam :
					fbFormat(sFormat := 'r%01d,', arg1 := F_BYTE(yChannel), sOut => sTempString);
					iOffsetCurrent := STRING_TO_INT(MID(sLastStringRec,5,4));
					iCurrentRatio := STRING_TO_INT(MID(sLastStringRec,5,10));
					IF (LEN(sLastStringRec) = 17) AND (LEFT(strReceived,3) = sTempString) THEN
						eStep := 1;
					ELSE
						eStep := 0; (* error *)
					END_IF
				MCRC_StartPower :
					fbFormat(sFormat := 'g%01d', arg1 := F_BYTE(yChannel), sOut => sTempString);
					IF (LEN(sLastStringRec) = 5) AND (LEFT(strReceived,2) = sTempString) THEN
						eStep := 1;
					ELSE
						eStep := 0; (* error *)
					END_IF
				MCRC_GetPower :
					fbFormat(sFormat := 'p%01d', arg1 := F_BYTE(yChannel), sOut => sTempString);
					IF (LEN(sLastStringRec) >= 13) THEN
						lrPower := STRING_TO_LREAL(MID(strReceived,7,4));
					ELSE
						bCommandError := TRUE;
					END_IF
				MCRC_SetSpeed :
					fbFormat(sFormat := 't%01d', arg1 := F_BYTE(yChannel), sOut => sTempString);
					IF (LEN(sLastStringRec) = 5) AND (LEFT(strReceived,2) = sTempString) THEN
						eStep := 1;
					ELSE
						eStep := 0; (* error *)
					END_IF
				MCRC_SetRatio :
					fbFormat(sFormat := 'd%01d', arg1 := F_BYTE(yChannel), sOut => sTempString);
					IF (LEN(sLastStringRec) = 5) AND (LEFT(strReceived,2) = sTempString) THEN
						eStep := 1;
					ELSE
						eStep := 0; (* error *)
					END_IF
				MCRC_UpdateMemory :
					sTempString := 'k';
					IF (LEN(sLastStringRec) = 4) AND (LEFT(strReceived,1) = sTempString) THEN
						eStep := 1;
					ELSE
						eStep := 0; (* error *)
					END_IF
				MCRC_DefineCurrentThr :
					fbFormat(sFormat := 'm%01d', arg1 := F_BYTE(yChannel), sOut => sTempString);
					IF (LEN(sLastStringRec) = 5) AND (LEFT(strReceived,2) = sTempString) THEN
						eStep := 1;
					ELSE
						eStep := 0; (* error *)
					END_IF
				MCRC_DefineMachineID :
					sTempString := 'x';
					IF (LEN(sLastStringRec) = 4) AND (LEFT(strReceived,1) = sTempString) THEN
						eStep := 1;
					ELSE
						eStep := 0; (* error *)
					END_IF
				MCRC_GetStatus :
					sTempString := 'z';
					IF (LEN(sLastStringRec) = 8) THEN
						ayChannelStatus[0] := STRING_TO_BYTE(MID(strReceived,2,2));
						ayChannelStatus[1] := STRING_TO_BYTE(MID(strReceived,2,4));
					ELSE
						bCommandError := TRUE;
					END_IF
			END_CASE
		ELSE
			eStep := 0;
		END_IF
		
		IF eStep = 0 THEN
			IF bFirstError THEN
				bFirstError := FALSE;
				eStep := 1;
			ELSE
				bCommandExecuted := TRUE;
			END_IF
		ELSE
			bCommandExecuted := TRUE;
		END_IF
		IF bCommandExecuted THEN
			bFirstError := TRUE;
			bCommandError := (eStep = 0);
			eStep := 1;
			eCommand := MCRC_None;
		END_IF
END_CASE

IF bWriteFile THEN
	fbWriteFile (
		sNetId			:=	'',
		hFile			:=	hLogFile,
		pWriteBuff		:=	ADR(acLogText),
		cbWriteLen		:=	INT_TO_UDINT(LEN(acLogText)),
		bExecute		:=	bCanLog
	);
	bCanLog := FALSE;
END_IF

IF bReset THEN
	bCommandError := FALSE;
END_IF

END_FUNCTION_BLOCK

// ---- POUs/utils/yCalcCheckSum.TcPOU
FUNCTION yCalcCheckSum : BYTE
VAR_INPUT
	sFrameWoChecksum	: STRING(255);
END_VAR
VAR
	i					: INT;
	yChecksum			: BYTE;
	size 					: INT;
	ps 					: POINTER TO BYTE;
	yData				: BYTE;
END_VAR

(* Sum the frame data *)
yChecksum := 0;
size := LEN(sFrameWoChecksum)-1;
ps := ADR(sFrameWoChecksum);
IF size>255 THEN size := 255; END_IF
FOR i:=0 TO size DO
	yData := ps^;
	yChecksum := yChecksum + yData;
	ps := ps + 1;
END_FOR

yChecksum := NOT yChecksum + 1;
yCalcCheckSum := yChecksum;

END_FUNCTION

// ---- POUs/utils/Dispersion.TcPOU
FUNCTION_BLOCK Dispersion
VAR_INPUT
	bGenerate		: BOOL;
	bNewPart		: BOOL;
	nPearl			: UINT;
END_VAR
VAR_OUTPUT
	lrDispersionX		: LREAL;
	lrDispersionY		: LREAL;
	lrDispersionZ		: LREAL;
END_VAR
VAR PERSISTENT
	iSeed			: INT := 0;
END_VAR
VAR
	CreateRandom				: DRAND;
	n							: uINT;
END_VAR

IF bNewPart THEN
	IF iSeed = 32767 THEN
		iSeed := -32768;
	ELSE
		iSeed := iSeed+1;
	END_IF
END_IF
IF bGenerate THEN
	(*Reinit random generator with current seed*)
	IF iSeed = 0 THEN
		CreateRandom( Seed := -1);
	ELSE
		CreateRandom( Seed := 0);
	END_IF
	CreateRandom( Seed := iSeed);

	FOR n := 0 TO nPearl * 3 DO
		CreateRandom( Seed := iSeed);
	END_FOR
	CreateRandom( Seed := iSeed , Num => lrDispersionX);
	CreateRandom( Seed := iSeed , Num => lrDispersionY);
	CreateRandom( Seed := iSeed , Num => lrDispersionZ);
END_IF

END_FUNCTION_BLOCK

// ---- POUs/Handlers/SharpenHdl.TcPOU
FUNCTION_BLOCK SharpenHdl

(*
	Description 	: Bloc fonction de gestion de l'affutage
	Auteur		: GRM
	Date		: 26.03.2014
	Version		: 1.00

	Modifications : 

*)

VAR_INPUT
	bEnable						: BOOL;
	bPowerOn					: BOOL;
	bResetErrors					: BOOL;
	bStopReq					: BOOL;
	bPauseReq					: BOOL;
	bPosTensioner				: BOOL;
	eCommand					: TModuleCommands;
	eRunCommand				: TRunCmdSharpen;
END_VAR
VAR_OUTPUT
	bModuleError					: BOOL;
	bSharpenAxisError			: BOOL;
	bNoTapeError				: BOOL;
	eRunStatus					: TRunStatus;
END_VAR
VAR_IN_OUT
	sSharpenAxis					: AXIS_REF;
	sSharpenEncoder				: AXIS_REF;
	sCurrentState					: TModuleData;
	TManualCmd					: TManSharpen;
END_VAR
VAR PERSISTENT
	lrSharpenMovePos			: LREAL					:= 10;
END_VAR
VAR CONSTANT
END_VAR
VAR
	lrSharpenTargetPos			: LREAL;
	eMoveSharpenAxisCommand	: TAxisCommands	:= AC_None;
	eMoveSharpenEncCommand	: TAxisCommands	:= AC_None;
	TSharpenAxis				: StdAxis;
	TSharpenEncoder				: StdAxis;
(*	eSaveStep					: TModuleSteps;*)
	lrCurrentSharpenMoveSpeed	: LREAL;
	DummyServoOn				: TManButton;
	TCheckNoTape				: TON;
END_VAR

IF (NOT sCurrentState.bStepMode) THEN
	sCurrentState.bWaitStep := FALSE;
END_IF

CASE eCommand OF
	MC_NoCmd :
		CASE sCurrentState.eStatus OF
			MS_Init :
				IF bEnable THEN
				CASE sCurrentState.eStep OF
					SP_InitStp1 : (* Init all synchros *)
						lrSharpenTargetPos := lrSharpenMovePos;
						sCurrentState.eStep := SP_InitStp2;
					SP_InitStp2 : (* Init sharpen tape axis *)
						eMoveSharpenAxisCommand := AC_Init;
						sCurrentState.eStep := SP_InitStp3;
					SP_InitStp3 :
						IF TSharpenAxis.eCurrentState = AS_InPosition THEN
							eMoveSharpenEncCommand := AC_ClearPosition;
							sCurrentState.eStep := SP_InitStp99;
						END_IF
					SP_InitStp99 : (* Leave Init *)
						sCurrentState.eStep := SP_RunStp1;
						sCurrentState.eStatus := MS_Ready;
						sCurrentState.bInitDone := TRUE;
				END_CASE
				ELSE
					sCurrentState.eStatus := MS_Ready;
					sCurrentState.bInitDone := TRUE;
				END_IF
			MS_Running :
				IF bEnable AND  (NOT sCurrentState.bWaitStep) THEN
					CASE sCurrentState.eStep OF
						SP_RunStp1 :(* Wait request *)
							eRunStatus := RS_WaitRequest;
							CASE eRunCommand OF
								RCS_None:
									IF bStopReq  THEN
										sCurrentState.eStatus := MS_Ready;
									ELSIF bPauseReq  THEN
										sCurrentState.eStatus := MS_Paused;
									END_IF
								RCS_MoveStep:
									sCurrentState.eStep := SP_RunStp10;
							END_CASE
							IF sCurrentState.eStep<> SP_RunStp1 THEN eRunStatus := RS_ProcessRequest1; END_IF
						SP_RunStp10 : (* Move one step *)
							eMoveSharpenAxisCommand := AC_MoveAtSpeed;
							TCheckNoTape(in := FALSE);
							sCurrentState.eStep := SP_RunStp11;
						SP_RunStp11 :
							TCheckNoTape(in := TRUE,pt := t#10s);
							IF (TSharpenEncoder.lrCurrentPos > lrSharpenMovePos) THEN
								eMoveSharpenAxisCommand := AC_Stop;
								sCurrentState.eStep := SP_RunStp12;
							ELSIF TCheckNoTape.Q THEN
								bNoTapeError := TRUE;
							END_IF
						SP_RunStp12 :
							IF (TSharpenAxis.eCurrentState = AS_InPosition) THEN
								eMoveSharpenEncCommand := AC_ClearPosition;
								sCurrentState.eStep := SP_RunStp1;
							END_IF
					END_CASE
				END_IF
			MS_Manual :
				TManualCmd.TSharpenAxis.Home.Enable := (TSharpenAxis.eCurrentState = AS_InPosition) OR (TSharpenAxis.eCurrentState = AS_NotHomed);
				TManualCmd.TSharpenAxis.MoveFw.Enable := TSharpenAxis.eCurrentState = AS_InPosition AND NOT bPosTensioner;
				TManualCmd.TSharpenAxis.CurrentPos := TSharpenAxis.lrCurrentPos;
				TManualCmd.bTapeNotEmpty := NOT bPosTensioner;
				TManualCmd.TMove2NextTapePos.Enable :=  TManualCmd.TSharpenAxis.MoveFw.Enable;
				CASE sCurrentState.eStep OF
					SP_ManualStp0 :
						 TManualCmd.lrStep := lrSharpenMovePos;
						TManualCmd.TSharpenAxis.JogStep := lrSharpenMovePos;
						TManualCmd.TSharpenAxis.MoveFw.Activate := FALSE;
						TManualCmd.TSharpenAxis.MoveBw.Activate := FALSE;
						TManualCmd.TSharpenAxis.Home.Activate := FALSE;
						TManualCmd.TMove2NextTapePos.Activate := FALSE;
						TManualCmd.TSharpenAxis.MoveBw.Enable := FALSE;
						sCurrentState.eStep := SP_ManualStp1;
					SP_ManualStp1 :
						IF bStopReq THEN
							sCurrentState.eStatus := MS_Stopped;
						ELSE
							IF TManualCmd.TMove2NextTapePos.Activate THEN
								lrSharpenTargetPos := lrSharpenMovePos;
								sCurrentState.eStep := SP_ManualStp10;
							END_IF
							IF (lrSharpenMovePos <> TManualCmd.lrStep) THEN
								lrSharpenMovePos :=  TManualCmd.lrStep;
							END_IF
							IF TManualCmd.TSharpenAxis.MoveFw.Activate THEN
								lrSharpenTargetPos := TManualCmd.TSharpenAxis.JogStep;
								sCurrentState.eStep := SP_ManualStp10;
							END_IF
							IF TManualCmd.TSharpenAxis.Home.Activate AND sCurrentState.eStep = SP_ManualStp1 THEN
								sCurrentState.eStep := SP_ManualStp20;
							END_IF
						END_IF
					SP_ManualStp10: (* Do the movement *)
						eMoveSharpenAxisCommand := AC_MoveAtSpeed;
						TCheckNoTape(in := FALSE);
						sCurrentState.eStep := SP_ManualStp11;
					SP_ManualStp11 :
						TCheckNoTape(in := TRUE,pt := t#10s);
						IF (TSharpenEncoder.lrCurrentPos > lrSharpenMovePos) THEN
							eMoveSharpenAxisCommand := AC_Stop;
							sCurrentState.eStep := SP_ManualStp12;
						ELSIF TCheckNoTape.Q THEN
							bNoTapeError := TRUE;
							sCurrentState.eStep := SP_ManualStp12;
						END_IF
					SP_ManualStp12 :(* Wait until position is reached *)
						CASE TSharpenAxis.eCurrentState OF
							AS_InPosition, AS_InError:
								eMoveSharpenEncCommand := AC_ClearPosition;
								TManualCmd.TMove2NextTapePos.Activate := FALSE;
								TManualCmd.TSharpenAxis.MoveFw.Activate := FALSE;
								sCurrentState.eStep := SP_ManualStp1;
						END_CASE
					SP_ManualStp20 : (* Init sharpen tape axis *)
						eMoveSharpenAxisCommand := AC_Home;
						sCurrentState.eStep := SP_ManualStp21;
					SP_ManualStp21 : (* Wait init done *)
						CASE TSharpenAxis.eCurrentState OF
							AS_InPosition, AS_InError:
								TManualCmd.TSharpenAxis.Home.Activate := FALSE;
								sCurrentState.eStep := SP_ManualStp1;
						END_CASE
				END_CASE
			MS_Paused:
				IF bStopReq THEN
					sCurrentState.eStatus := MS_Ready;
				END_IF
		END_CASE
	MC_Init :
		IF sCurrentState.bInitDone  THEN
			sCurrentState.eStep := SP_InitStp99;
		ELSE
			sCurrentState.eStep := SP_InitStp1;
		END_IF
		sCurrentState.eStatus := MS_Init;
	MC_Run :
		sCurrentState.eStatus := MS_Running;
	MC_Manual :
		sCurrentState.bInitDone := FALSE;
		sCurrentState.eStatus := MS_Manual;
		sCurrentState.eStep := SP_ManualStp0;
	MC_Stop :
		sCurrentState.eStatus := MS_Stopped;
END_CASE;

IF bResetErrors THEN
	bNoTapeError := FALSE;
	sCurrentState.bInError := FALSE;
END_IF

IF bPosTensioner THEN
	bNoTapeError 	:= TRUE;
END_IF

IF bNoTapeError AND TSharpenAxis.eCurrentState = AS_Moving  THEN
	eMoveSharpenAxisCommand := AC_ForceStop;
END_IF

(* Sharpen Axis *)
IF (sCurrentState.eStatus = MS_Manual) THEN
	lrCurrentSharpenMoveSpeed := TSharpenAxis.lrManualSpeed;
ELSE
	lrCurrentSharpenMoveSpeed := TSharpenAxis.lrRunningSpeed;
END_IF
TSharpenAxis(
	eCommand		:= eMoveSharpenAxisCommand ,
	lrTargetPos		:= lrSharpenTargetPos ,
	lrTargetSpeed	:= lrCurrentSharpenMoveSpeed ,
	bResetErrors		:= bResetErrors ,
	bPowerIsOn		:= bPowerOn ,
	eHomingAxisType:= AHT_NoHoming ,
	bNegLimitSwitch	:= TRUE,  (* cannot go backward *)
	sAxis			:= sSharpenAxis,
	stServoButton 	:= TManualCmd.TSharpenAxis.ServoON
);
eMoveSharpenAxisCommand := AC_None;
bSharpenAxisError := (TSharpenAxis.eCurrentState = AS_InError);
TSharpenEncoder(
	eCommand		:= eMoveSharpenEncCommand ,
	lrTargetPos		:= 0 ,
	lrTargetSpeed	:= 0 ,
	bResetErrors		:= bResetErrors ,
	bPowerIsOn		:= FALSE ,
	eHomingAxisType:= AHT_NoHoming ,
	sAxis			:= sSharpenEncoder,
	stServoButton 	:= DummyServoOn
);
eMoveSharpenEncCommand := AC_None;

IF NOT bEnable THEN
	bModuleError := FALSE;
	bSharpenAxisError := FALSE;
	bNoTapeError := FALSE;
END_IF

IF NOT bPowerOn OR bSharpenAxisError OR bNoTapeError THEN
	sCurrentState.bInError := TRUE;
		IF (sCurrentState.eStatus <> MS_Manual) AND (sCurrentState.eStatus <> MS_Stopped) AND (sCurrentState.eStatus <> MS_Init) THEN
		sCurrentState.eStatus := MS_Ready;
	END_IF
END_IF

IF NOT bPowerOn OR bSharpenAxisError THEN
	sCurrentState.bInitDone := FALSE;
	IF (sCurrentState.eStatus <> MS_Manual) THEN
		sCurrentState.eStatus := MS_Stopped;
	END_IF
END_IF

bModuleError := sCurrentState.bInError;
sCurrentState.bRunning := (sCurrentState.eStatus = MS_Running);
IF (sCurrentState.eStatus <> MS_Running) THEN eRunStatus := RS_NotRunning; END_IF

END_FUNCTION_BLOCK

// ---- POUs/Handlers/TurnOverHdl.TcPOU
FUNCTION_BLOCK TurnOverHdl

(*
	Description 	: Bloc fonction de gestion du retourneur
	Auteur		: GRM
	Date		: 26.03.2014
	Version		: 1.00

	Modifications :

*)

VAR_INPUT
	bEnable						: BOOL;
	bPowerOn					: BOOL;
	bResetErrors					: BOOL;
	bIndexTurnOver				: BOOL;
	bFixVacuumOk				: BOOL;
	bArmVacuumOk				: BOOL;
	bJackIsDown					: BOOL;
	bJackIsUp					: BOOL;
	bStopReq					: BOOL;
	bPauseReq					: BOOL;
	eCommand					: TModuleCommands;
	eRunCommand				:TRunCmdTurnOver;
	sInGiveToLoader				: TTaker;
	sInTakeFromLoader			: TGiver;
	bManInterlock				: BOOL;
	sVaccumSettings				: TVaccumSettings;
END_VAR
VAR_OUTPUT
	bModuleError					: BOOL;
	bJackError					: BOOL;
	bArmVacuumError				: BOOL;
	bFixVacuumError				: BOOL;
	bTurnOverAxisError			: BOOL;
	bMoveJackDown				: BOOL;
	bMoveJackUp				: BOOL;
	bActivateArmVacuum			: BOOL;
	bActivateArmBlowing			: BOOL;
	bActivateFixVacuum			: BOOL;
	bActivateFixBlowing			: BOOL;
	bActivateCleaningBlow			: BOOL;
	eRunStatus					: TRunStatus;
	sOutGiveToLoader			: TGiver;
	sOutTakeFromLoader			: TTaker;
	sRunData					: TRunDataTurnOver;
	bManInterlockOut				: BOOL;
END_VAR
VAR_IN_OUT
	sCurrentState					: TModuleData;
	TManualCmd					: TManTurnOver;
	sTurnOverAxisRef				: AXIS_REF;
END_VAR
VAR CONSTANT
	lrSafeTolerance 				:LREAL 					:= 1;			(* Tolerance for safety axis *)
END_VAR
VAR PERSISTENT
	lrTurnOverIndexPos			: LREAL					:= 0;			(* Positionnement du retourneur en position attente *)
	lrTurnOverFlippedPos			: LREAL					:= 180;		(* Positionnement du retourneur en position retourné *)
	lrTurnOverJogStep			: LREAL					:= 1;
END_VAR
VAR
	bEnableArmVacuum			: BOOL;
	bEnableFixVacuum			: BOOL;
	bDisableArmVacuumChecking	: BOOL;
	bDisableFixVacuumChecking	: BOOL;
	eMoveTurnOverAxisCommand	: TAxisCommands	:= AC_None;
	lrTurnOverTargetPos			: LREAL;
	TTurnOverAxis				: StdAxis;
	TJack						: FB_CheckJack2_2;
	TArmVacuum					: FB_Vacuum;
	TFixVacuum					: FB_Vacuum;
	lrCurrentTurnOverMoveSpeed	: LREAL;
	TCleanFixTimer				: TON;
	TVacuumTimer				: TON;
	eLastStatus 					: TModuleStatus := MS_Stopped;
END_VAR

IF (NOT sCurrentState.bStepMode) THEN
	sCurrentState.bWaitStep := FALSE;
END_IF

IF eLastStatus<>sCurrentState.eStatus THEN
	IF eLastStatus=MS_Manual THEN
		(*Leave manual mode, redefine part present base on vacuum *)
		IF NOT bActivateArmVacuum THEN
			sRunData.aTPartData[TO_Arm].bPartPresent := FALSE;
		END_IF
		IF NOT bEnableFixVacuum THEN
			sRunData.aTPartData[TO_Fix].bPartPresent := FALSE;
		END_IF
	END_IF
	IF eLastStatus=MS_Running OR sCurrentState.eStatus=MS_Manual THEN
		(* Set vaccum base on part present, Vacuum can be disable if take part has failed*)
		bActivateArmVacuum := sRunData.aTPartData[TO_Arm].bPartPresent;
		bEnableFixVacuum := sRunData.aTPartData[TO_Fix].bPartPresent;
	END_IF
	eLastStatus := sCurrentState.eStatus;
END_IF

CASE eCommand OF
	MC_NoCmd :
		CASE sCurrentState.eStatus OF
			MS_Init :
				CASE sCurrentState.eStep OF
					SP_InitStp1 :
						IF bEnable THEN
							bActivateCleaningBlow := FALSE;
							bDisableArmVacuumChecking := FALSE;
							bDisableFixVacuumChecking := FALSE;
							TVacuumTimer(IN := FALSE);
							(*bActivateArmVacuum := TRUE;
							bEnableFixVacuum := TRUE;*)
							sCurrentState.eStep := SP_InitStp2;
						ELSE
							sCurrentState.eStep := SP_InitStp99;
						END_IF
					SP_InitStp2 :
						TVacuumTimer(IN := TRUE, PT := t#0s);
						IF TVacuumTimer.Q THEN
							(* Check where there is parts *)
							(*IF TArmVacuum.bVacuumCorrect THEN sRunData.aTPartData[TO_Arm].bPartPresent := TRUE; END_IF
							IF TFixVacuum.bVacuumCorrect THEN sRunData.aTPartData[TO_Fix].bPartPresent := TRUE; END_IF*)
							bActivateArmVacuum := sRunData.aTPartData[TO_Arm].bPartPresent;
							bEnableFixVacuum := sRunData.aTPartData[TO_Fix].bPartPresent;
							IF sCurrentState.bInitDone THEN
								sCurrentState.eStep := SP_InitStp99;
							ELSE
								sCurrentState.eStep := SP_InitStp3;
							END_IF
						END_IF
					SP_InitStp3 : (* Lower the jack *)
						bMoveJackUp := FALSE;
						sCurrentState.eStep := SP_InitStp4;
					SP_InitStp4 : (* Check if jack is up *)
						IF bJackIsDown THEN
							sCurrentState.eStep := SP_InitStp5;
						END_IF
					SP_InitStp5 : (* Init turn over axis *)
						eMoveTurnOverAxisCommand := AC_Init;
						sCurrentState.eStep := SP_InitStp6;
					SP_InitStp6 : (* Rotate the turn over to go to index position *)
						IF TTurnOverAxis.eCurrentState = AS_InPosition THEN
							lrTurnOverTargetPos := lrTurnOverIndexPos;
							eMoveTurnOverAxisCommand := AC_MoveAtAbsPos;
							sCurrentState.eStep := SP_InitStp7;
						END_IF
					SP_InitStp7 : (* Wait until index position is reached *)
						IF TTurnOverAxis.eCurrentState = AS_InPosition THEN
							sCurrentState.eStep := SP_InitStp99;
						END_IF
					SP_InitStp99 : (* Leave Init *)
						sCurrentState.eStep := SP_RunStp1;
						sCurrentState.eStatus := MS_Ready;
						sCurrentState.bInitDone := TRUE;
				END_CASE
			MS_Running :
				IF (NOT sCurrentState.bWaitStep) THEN
					CASE sCurrentState.eStep OF
						SP_RunStp1 :
							eRunStatus := RS_WaitRequest;
							IF bEnable THEN
								CASE eRunCommand OF
									RCTO_None:
										IF bStopReq  THEN
											sCurrentState.eStatus := MS_Ready;
										ELSIF bPauseReq  THEN
											sCurrentState.eStatus := MS_Paused;
										END_IF
									RCTO_TakePart:
										sOutTakeFromLoader.bReadyToTake := FALSE;
										sOutTakeFromLoader.bHasTaken := FALSE;
										sCurrentState.eStep := SP_RunStp10;
									RCTO_GivePart:
										sOutGiveToLoader.bHasGiven := FALSE;
										sOutGiveToLoader.bPartDataReady := FALSE;
										sCurrentState.eStep := SP_RunStp20;
									RCTO_Turn:
										sCurrentState.eStep := SP_RunStp30;
								END_CASE
							ELSE
								IF bStopReq  THEN
									sCurrentState.eStatus := MS_Ready;
								ELSIF bPauseReq  THEN
									sCurrentState.eStatus := MS_Paused;
								END_IF
							END_IF
							IF sCurrentState.eStep<> SP_RunStp1 THEN eRunStatus := RS_ProcessRequest1; END_IF
						SP_RunStp10 :  (*Take Part*)
							IF sInTakeFromLoader.bPartDataReady THEN
								sRunData.aTPartData[TO_Arm] := sInTakeFromLoader.TPartData;
								sRunData.aTPartData[TO_Arm].bPartPresent := FALSE;
								sCurrentState.eStep := SP_RunStp11;
							END_IF
						SP_RunStp11 :
							bEnableArmVacuum := TRUE;
							bDisableArmVacuumChecking := TRUE;
							sOutTakeFromLoader.bReadyToTake := TRUE;
							sCurrentState.eStep := SP_RunStp12;
						SP_RunStp12 :
							(* Wait until left loader has given *)
							IF sInTakeFromLoader.bHasGiven THEN
								bDisableArmVacuumChecking := FALSE;
								sCurrentState.eStep := SP_RunStp13;
							END_IF
						SP_RunStp13 :
							(* Check if the part is on arm *)
							IF TArmVacuum.bVacuumCorrect THEN
								sOutTakeFromLoader.bHasTaken := TRUE;
								sRunData.aTPartData[TO_Arm].bPartPresent := TRUE;
								sCurrentState.eStep := SP_RunStp1;
							END_IF
						SP_RunStp20 : (*Give Part*)
							sOutGiveToLoader.TPartData := sRunData.aTPartData[TO_Fix];
							sOutGiveToLoader.bPartDataReady := TRUE;
							sCurrentState.eStep := SP_RunStp21;
						SP_RunStp21 :
							IF sInGiveToLoader.bReadyToTake THEN
								bEnableFixVacuum := FALSE;
								sCurrentState.eStep := SP_RunStp22;
							END_IF
						SP_RunStp22 :
							(* Check if laying vacuum is disabled *)
							IF TFixVacuum.bVacuumCorrect THEN
								sOutGiveToLoader.bHasGiven := TRUE;
								sCurrentState.eStep := SP_RunStp23;
							END_IF
						SP_RunStp23 :
							(* Check if right loader has taken the plate *)
							IF sInGiveToLoader.bHasTaken THEN
								sRunData.aTPartData[TO_Fix].bPartPresent := FALSE;
								sCurrentState.eStep := SP_RunStp1;
							END_IF
						SP_RunStp30 : (*TurnOver *)
							bActivateCleaningBlow := TRUE;
							TCleanFixTimer(IN:=FALSE);
							sCurrentState.eStep := SP_RunStp31;
						SP_RunStp31 :
							TCleanFixTimer(IN :=TRUE,PT := t#1s);
							IF TCleanFixTimer.Q THEN
								bActivateCleaningBlow := FALSE;
								sCurrentState.eStep := SP_RunStp32;
							END_IF
						SP_RunStp32 :
							lrTurnOverTargetPos := lrTurnOverFlippedPos;
							eMoveTurnOverAxisCommand := AC_MoveAtAbsPos;
							sCurrentState.eStep := SP_RunStp33;
						SP_RunStp33 :
							(* Wait until flip position is reached - Raise Jack *)
							IF TTurnOverAxis.eCurrentState = AS_InPosition THEN
								bMoveJackUp := TRUE;
								sCurrentState.eStep := SP_RunStp34;
							END_IF
						SP_RunStp34 :
							(* Check if jack is up - Enable laying vacuum and disable manipulator vacuum *)
							IF bJackIsUp THEN
								sRunData.aTPartData[TO_Fix] := sRunData.aTPartData[TO_Arm];
								sRunData.aTPartData[TO_Fix].ePartSide := PS_SOUS;
								bEnableFixVacuum := TRUE;
								bEnableArmVacuum := FALSE;
								sCurrentState.eStep := SP_RunStp35;
							END_IF
						SP_RunStp35 :
							(* Wait until laying vacuum is OK - Lower Jack *)
							IF TFixVacuum.bVacuumCorrect AND TArmVacuum.bVacuumCorrect THEN
								sRunData.aTPartData[TO_Arm].bPartPresent := FALSE;
								bMoveJackUp := FALSE;
								sCurrentState.eStep := SP_RunStp36;
							END_IF
						SP_RunStp36 :
							(* Check if jack is Down - Flip back the turn over *)
							IF bJackIsDown THEN
								lrTurnOverTargetPos := lrTurnOverIndexPos;
								eMoveTurnOverAxisCommand := AC_MoveAtAbsPos;
								sCurrentState.eStep := SP_RunStp37;
							END_IF
						SP_RunStp37 :
							(* Wait until index position is reached *)
							IF TTurnOverAxis.eCurrentState = AS_InPosition THEN
								sCurrentState.eStep := SP_RunStp1;
							END_IF
					END_CASE
				END_IF
			MS_Manual :
				TManualCmd.TJack.Enable := TRUE;
				TManualCmd.TTurnOverAxis.Home.Enable := NOT bManInterlock AND (TTurnOverAxis.eCurrentState = AS_InPosition) OR (TTurnOverAxis.eCurrentState = AS_NotHomed);
				TManualCmd.TTurnOverAxis.MoveBw.Enable := NOT bManInterlock AND (TTurnOverAxis.eCurrentState = AS_InPosition) AND (TTurnOverAxis.lrCurrentPos-lrTurnOverJogStep >= TTurnOverAxis.lrMinPos);
				TManualCmd.TTurnOverAxis.MoveFw.Enable := NOT bManInterlock AND (TTurnOverAxis.eCurrentState = AS_InPosition) AND (TTurnOverAxis.lrCurrentPos+lrTurnOverJogStep <= TTurnOverAxis.lrMaxPos);
				TManualCmd.TTurnOverAxisIndexPos.MoveToTeach.Enable := NOT bManInterlock AND (TTurnOverAxis.eCurrentState = AS_InPosition) AND lrTurnOverIndexPos >= TTurnOverAxis.lrMinPos AND lrTurnOverIndexPos <= TTurnOverAxis.lrMaxPos;
				TManualCmd.TTurnOverAxisFlippedPos.MoveToTeach.Enable := NOT bManInterlock AND (TTurnOverAxis.eCurrentState = AS_InPosition) AND lrTurnOverFlippedPos >= TTurnOverAxis.lrMinPos AND lrTurnOverFlippedPos <= TTurnOverAxis.lrMaxPos;
				TManualCmd.TTurnOverAxis.CurrentPos := TTurnOverAxis.lrCurrentPos;
				TManualCmd.TActivateFixVacuum.Enable := TTurnOverAxis.eCurrentState <> AS_Moving AND TTurnOverAxis.eCurrentState <> AS_Stopping AND TTurnOverAxis.eCurrentState <> AS_Homing;
				TManualCmd.TActivateArmVacuum.Enable := TManualCmd.TActivateFixVacuum.Enable;
				TManualCmd.TTurnOverAxisIndexPos.TeachedPos := lrTurnOverIndexPos;
				TManualCmd.TTurnOverAxisFlippedPos.TeachedPos := lrTurnOverFlippedPos;
				bManInterlockOut := NOT ((TTurnOverAxis.lrCurrentPos <= (lrTurnOverIndexPos+lrSafeTolerance)) AND
								TTurnOverAxis.bAxisHomed);

				CASE sCurrentState.eStep OF
					SP_ManualStp0 :
						TManualCmd.TTurnOverAxis.JogStep := lrTurnOverJogStep;
						TManualCmd.TTurnOverAxis.MoveBw.Activate := FALSE;
						TManualCmd.TTurnOverAxis.MoveFw.Activate := FALSE;
						TManualCmd.TTurnOverAxisIndexPos.MoveToTeach.Activate := FALSE;
						TManualCmd.TTurnOverAxisIndexPos.Teach := FALSE;
						TManualCmd.TTurnOverAxisFlippedPos.MoveToTeach.Activate := FALSE;
						TManualCmd.TTurnOverAxisFlippedPos.Teach := FALSE;
						TManualCmd.TActivateFixVacuum.Activate := bEnableFixVacuum;
						TManualCmd.TActivateArmVacuum.Activate := bEnableArmVacuum;
						TManualCmd.TJack.Activate := bMoveJackUp;
						TManualCmd.TTurnOverAxis.Home.Activate := FALSE;
						TManualCmd.TActivateCleaningBlow.Enable := TRUE;
						TManualCmd.TActivateCleaningBlow.Activate := bActivateCleaningBlow;
						sCurrentState.eStep := SP_ManualStp1;
					SP_ManualStp1:
						IF bStopReq THEN
							sCurrentState.eStatus := MS_Stopped;
						ELSE
							IF (lrTurnOverJogStep <> TManualCmd.TTurnOverAxis.JogStep) THEN
								lrTurnOverJogStep := TManualCmd.TTurnOverAxis.JogStep;
							END_IF
							IF TManualCmd.TTurnOverAxisIndexPos.Teach THEN
								lrTurnOverIndexPos := TTurnOverAxis.lrCurrentPos;
								TManualCmd.TTurnOverAxisIndexPos.Teach := FALSE;
							END_IF
							IF TManualCmd.TTurnOverAxisIndexPos.MoveToTeach.Activate THEN
								lrTurnOverTargetPos := TManualCmd.TTurnOverAxisIndexPos.TeachedPos;
								sCurrentState.eStep := SP_ManualStp10;
							END_IF
							IF TManualCmd.TTurnOverAxisFlippedPos.Teach THEN
								lrTurnOverFlippedPos := TTurnOverAxis.lrCurrentPos;
								TManualCmd.TTurnOverAxisFlippedPos.Teach := FALSE;
							END_IF
							IF TManualCmd.TTurnOverAxisFlippedPos.MoveToTeach.Activate THEN
								lrTurnOverTargetPos := TManualCmd.TTurnOverAxisFlippedPos.TeachedPos;
								sCurrentState.eStep := SP_ManualStp10;
							END_IF
							IF TManualCmd.TTurnOverAxis.MoveBw.Activate THEN
								lrTurnOverTargetPos := TTurnOverAxis.lrCurrentPos - lrTurnOverJogStep;
								sCurrentState.eStep := SP_ManualStp10;
							END_IF
							IF TManualCmd.TTurnOverAxis.MoveFw.Activate THEN
								lrTurnOverTargetPos := TTurnOverAxis.lrCurrentPos + lrTurnOverJogStep;
								sCurrentState.eStep := SP_ManualStp10;
							END_IF
							IF TManualCmd.TTurnOverAxis.Home.Activate AND sCurrentState.eStep = SP_ManualStp1 THEN
								sCurrentState.eStep := SP_ManualStp20;
							END_IF
							bEnableFixVacuum := TManualCmd.TActivateFixVacuum.Activate;
							bEnableArmVacuum := TManualCmd.TActivateArmVacuum.Activate;
						END_IF
					SP_ManualStp10: (* Do the movement *)
						eMoveTurnOverAxisCommand := AC_MoveAtAbsPos;
						sCurrentState.eStep := SP_ManualStp11;
					SP_ManualStp11: (* Wait until position is reached *)
						CASE TTurnOverAxis.eCurrentState OF
							AS_InPosition, AS_InError:
								TManualCmd.TTurnOverAxisIndexPos.MoveToTeach.Activate := FALSE;
								TManualCmd.TTurnOverAxisFlippedPos.MoveToTeach.Activate := FALSE;
								TManualCmd.TTurnOverAxis.MoveFw.Activate := FALSE;
								TManualCmd.TTurnOverAxis.MoveBw.Activate := FALSE;
								sCurrentState.eStep := SP_ManualStp1;
						END_CASE
					SP_ManualStp20 : (* Init turn over axis *)
						eMoveTurnOverAxisCommand := AC_Home;
						sCurrentState.eStep := SP_ManualStp21;
					SP_ManualStp21 : (* Rotate the turn over to go to index position *)
						CASE TTurnOverAxis.eCurrentState OF
							AS_InPosition:
								lrTurnOverTargetPos := lrTurnOverIndexPos;
								eMoveTurnOverAxisCommand := AC_MoveAtAbsPos;
								sCurrentState.eStep := SP_ManualStp22;
							AS_InError:
								sCurrentState.eStep := SP_ManualStp1;
								TManualCmd.TTurnOverAxis.Home.Activate := FALSE;
						END_CASE
					SP_ManualStp22 : (* Wait until index position is reached *)
						CASE TTurnOverAxis.eCurrentState OF
							AS_InPosition, AS_InError:
								sCurrentState.eStep := SP_ManualStp1;
								TManualCmd.TTurnOverAxis.Home.Activate := FALSE;
						END_CASE
				END_CASE
				bMoveJackUp := TManualCmd.TJack.Activate;
				bActivateCleaningBlow := TManualCmd.TActivateCleaningBlow.Activate;
			MS_Paused:
				IF bStopReq THEN
					sCurrentState.eStatus := MS_Ready;
				END_IF
		END_CASE
	MC_Init :
		sCurrentState.eStep := SP_InitStp1;
		sCurrentState.eStatus := MS_Init;
	MC_Run :
		sCurrentState.eStatus := MS_Running;
	MC_Manual :
		sCurrentState.bInitDone := FALSE;
		sCurrentState.eStatus := MS_Manual;
		sCurrentState.eStep := SP_ManualStp0;
	MC_Stop :
		sCurrentState.eStatus := MS_Stopped;
END_CASE;

IF bResetErrors THEN
	sCurrentState.bInError := FALSE;
END_IF

IF bEnable THEN
	(* Turn Over Axis *)
	IF (sCurrentState.eStatus = MS_Manual) THEN
		lrCurrentTurnOverMoveSpeed := TTurnOverAxis.lrManualSpeed;
	ELSE
		lrCurrentTurnOverMoveSpeed := TTurnOverAxis.lrRunningSpeed;
	END_IF
	TTurnOverAxis(
		eCommand		:= eMoveTurnOverAxisCommand,
		lrTargetPos		:= lrTurnOverTargetPos,
		lrTargetSpeed	:= lrCurrentTurnOverMoveSpeed,
		sAxis			:= sTurnOverAxisRef,
		bResetErrors		:= bResetErrors,
		bHomeSensor	:= bIndexTurnOver,
		bPowerIsOn		:= bPowerOn,
		stServoButton 	:= TManualCmd.TTurnOverAxis.ServoON
	);
	
	eMoveTurnOverAxisCommand := AC_None;
	bTurnOverAxisError := (TTurnOverAxis.eCurrentState = AS_InError);
	
	(* Check Jack Error *)
	bMoveJackDown := NOT bMoveJackUp;
	TJack(
		bJackGoIn	:= bMoveJackDown,
		bJackGoOut	:= bMoveJackUp,
		bJackIsIn	:= bJackIsDown,
		bJackIsOut	:= bJackIsUp,
		tTimeOut		:= t#2s,
		bResetErrors	:= bResetErrors,
		bJackError	=> bJackError
	 );
	
	(* Handle Manipulator Vacuum *)
	TArmVacuum(
		bEnableVacuum	:= bEnableArmVacuum,
		tVacErrorDelay		:= INT_TO_TIME(sVaccumSettings.iErrorDelay),
		tBlowingTime			:= INT_TO_TIME(sVaccumSettings.iBlowing),
		tWaitVacuumOK		:= INT_TO_TIME(sVaccumSettings.iWaitWhenVacuumOk),
		bReset			:= bResetErrors,
		bVacuumOK		:= bArmVacuumOk AND bEnableArmVacuum,
		bDisableVacuumChecking := bDisableArmVacuumChecking,
		bVacuumError	=> bArmVacuumError,
		bVacuumOn		=> bActivateArmVacuum,
		bBlowOn			=> bActivateArmBlowing,
	);
	
	(* Handle Laying Vacuum *)
	TFixVacuum(
		bEnableVacuum	:= bEnableFixVacuum,
		tVacErrorDelay		:= INT_TO_TIME(sVaccumSettings.iErrorDelay),
		tBlowingTime			:= INT_TO_TIME(sVaccumSettings.iBlowing),
		tWaitVacuumOK		:= INT_TO_TIME(sVaccumSettings.iWaitWhenVacuumOk),
		bReset			:= bResetErrors,
		bVacuumOK		:= bFixVacuumOk,
		bDisableVacuumChecking := bDisableFixVacuumChecking,
		bVacuumError	=> bFixVacuumError,
		bVacuumOn		=> bActivateFixVacuum,
		bBlowOn			=> bActivateFixBlowing,
	);
END_IF

IF NOT bPowerOn OR bTurnOverAxisError OR bJackError OR bArmVacuumError OR bFixVacuumError THEN
	sCurrentState.bInError := TRUE;
	IF (sCurrentState.eStatus <> MS_Manual) AND (sCurrentState.eStatus <> MS_Stopped) AND (sCurrentState.eStatus <> MS_Init) THEN
		sCurrentState.eStatus := MS_Ready;
	END_IF
END_IF

IF (NOT bPowerOn OR bTurnOverAxisError) THEN
	sCurrentState.bInitDone := FALSE;
	IF (sCurrentState.eStatus <> MS_Manual) THEN
		sCurrentState.eStatus := MS_Stopped;
	END_IF
END_IF

IF sCurrentState.eStatus <> MS_Running AND sCurrentState.eStatus <> MS_Manual  THEN
	bActivateCleaningBlow := FALSE;
END_IF

sCurrentState.bInterlocked := bManInterlock AND  (sCurrentState.eStatus = MS_Manual);
bModuleError := sCurrentState.bInError;
sCurrentState.bRunning := (sCurrentState.eStatus = MS_Running);
IF (sCurrentState.eStatus <> MS_Running) THEN eRunStatus := RS_NotRunning; END_IF

END_FUNCTION_BLOCK

// ---- POUs/Handlers/BarrelHdl.TcPOU
FUNCTION_BLOCK BarrelHdl

(*
	Description 	: Bloc fonction de gestion du barillet
	Auteur		: GRM
	Date		: 26.03.2014
	Version		: 1.00

	Modifications :

*)

VAR_INPUT
	bEnable						: BOOL;
	bNewJob					: BOOL;
	bJackIsDown					: BOOL;
	bJackIsUp					: BOOL;
	bPowerOn					: BOOL;
	bResetErrors					: BOOL;
	bStickPresent					: BOOL;
	bTableIndexed				: BOOL;
	bTableNotIndexed			: BOOL;
	bStopReq					: BOOL;
	bPauseReq					: BOOL;
	eCommand					: TModuleCommands;
	iStickArea					: INT;
	iStickUsedSection1			: INT;
	iStickUsedSection2			: INT;
	bSection1IsUsed				: BOOL;
	bSection2IsUsed				: BOOL;
	sInStickTake					: TTaker;
	eRunCommand				: TRunCmdBarrel;
	bManInterlock				: BOOL;
END_VAR
VAR_OUTPUT
	bModuleError					: BOOL;
	bBarrelAxisError				: BOOL;
	bArea1StickWarning			: BOOL;
	bArea2StickWarning			: BOOL;
	bArea3StickWarning			: BOOL;
	bArea4StickWarning			: BOOL;
	bJackError					: BOOL;
	bIndexError					: BOOL;
	bBarrelEmptyError				: BOOL;
	bMoveJackUp				: BOOL;
	bIndexTable					: BOOL;
	sOutStickTake				: TGiver;
	eRunStatus					: TRunStatus;
END_VAR
VAR_IN_OUT
	sCurrentState					: TModuleData;
	TManualCmd					: TManBarrel;
	sBarrelAxisRef				: AXIS_REF;
END_VAR
VAR PERSISTENT
	lrBarrelTakenPos				: LREAL					:= 53;			(* Position du premier bâtonnet devant l'ejecteur *)
	lrBarrelCheckPos				: LREAL					:= 270;			(* Position du premier bâtonnet devant le capteur *)
	lrBarrelJogStep				: LREAL					:= 7.5;
END_VAR
VAR CONSTANT
	iMaxPosition 					: INT := 11;
	iMaxSection 					:INT := 4;
	alrIndexSectionPosition		: ARRAY[1..iMaxSection,1..iMaxPosition] OF LREAL :=
										    [7.5,    15,   22.5,   30,    37.5,   45,   52.5,    60,   67.5,   75,   82.5,   (* section A *)
										  97.5, 105, 112.5, 120, 127.5, 135, 142.5, 150, 157.5, 165, 172.5,  (* section B *)
										187.5, 195, 202.5, 210, 217.5, 225, 232.5, 240, 247.5, 255, 262.5,  (* section C *)
										277.5, 285, 292.5, 300, 307.5, 315, 322.5, 330, 337.5, 345, 352.5];  (* section D *)
END_VAR
VAR
	i							: INT;
	j							: INT;
	bStickFound					: BOOL;
	bStartTimer					: BOOL					:= FALSE;
	bCommandError				: BOOL					:= FALSE;
	bBarrelNeedScan				: BOOL					:= FALSE;
	eMoveBarrelAxisCommand		: TAxisCommands	:= AC_None;
	lrBarrelTargetPos				: LREAL;
	lrCurrentBarrelMoveSpeed		: LREAL;
	TBarrelAxis					: StdAxis;
	TBarrelDetectionTimer			: TON;
	TJack						: FB_CheckJack1_2;
	TTableIndex					: FB_CheckJack1_2;
	iIndexPosition					: INT := 1;
	iIndexSection					: INT := 1;
	yMultiSection2Use				: BYTE := 1;
	iScanPearling				: INT := 0;
	iSearchIndexPosition			: INT := 1;
	iSearchIndexSection			: INT := 1;
	abStickPresent				: ARRAY[1..2,1..iMaxSection,1..iMaxPosition] OF BOOL :=
										    [FALSE, FALSE, FALSE, FALSE, FALSE, FALSE, FALSE, FALSE, FALSE, FALSE, FALSE, (* section A *)
										    FALSE, FALSE, FALSE, FALSE, FALSE, FALSE, FALSE, FALSE, FALSE, FALSE, FALSE, (* section B *)
										    FALSE, FALSE, FALSE, FALSE, FALSE, FALSE, FALSE, FALSE, FALSE, FALSE, FALSE, (* section C *)
										    FALSE, FALSE, FALSE, FALSE, FALSE, FALSE, FALSE, FALSE, FALSE, FALSE, FALSE]; (* section D *)
END_VAR

IF (NOT sCurrentState.bStepMode) THEN
	sCurrentState.bWaitStep := FALSE;
END_IF

IF NOT bSection1IsUsed THEN
	iStickUsedSection1 := 0;
END_IF
IF NOT bSection2IsUsed THEN
	iStickUsedSection2 := 0;
END_IF

